// TIA Portal V17 export
// export: Created 2025-03-07T09:18:09.3594696Z, ExportSetting WithDefaults, DisplayName Totally Integrated Automation Portal, DisplayVersion V17 Update 8, DisplayName TIA Portal Openness, DisplayVersion V17 Update 8, DisplayName TIA Portal Version Control Interface, DisplayVersion V17, DisplayName SINAMICS Startdrive Advanced, DisplayVersion V17 SP2, DisplayName SINAMICS Startdrive G110M, G120, G120C, G120D, G120P, G115D, DisplayVersion V17 SP2, DisplayName SINAMICS Startdrive G130, G150, S120, S150, SINAMICS MV, S210, DisplayVersion V17 SP2, DisplayName STEP 7 Professional, DisplayVersion V17 Update 8, DisplayName SINUMERIK ONE STEP 7 Toolbox, DisplayVersion V17 Update 12, DisplayName SINUMERIK 840D sl STEP 7 Toolbox, DisplayVersion V17 Update 12, DisplayName STEP 7 Safety, DisplayVersion V17 Update 6, DisplayName WinCC Advanced, DisplayVersion V17 Update 8
FUNCTION "FC1251_PART_CYCLE_UNIT_02_CLADDING" : Void   // FC1251, LAD
{ S7_Optimized_Access := 'FALSE' }
AUTHOR : ETXETAR
VERSION : 1.0
// stored: AutoNumber false, IsIECCheckEnabled false, SetENOAutomatically false, UDAEnableTagReadback false
   VAR CONSTANT
      FC_NUMBER : DInt := 1251;
   END_VAR
   VAR_TEMP   // added for the SCL form of the ladder/FBD networks
      _w1 : Bool;
      _w2 : Bool;
      _w3 : Bool;
      _w4 : Bool;
   END_VAR
BEGIN

REGION Network 1: GENERAL CONDITIONS
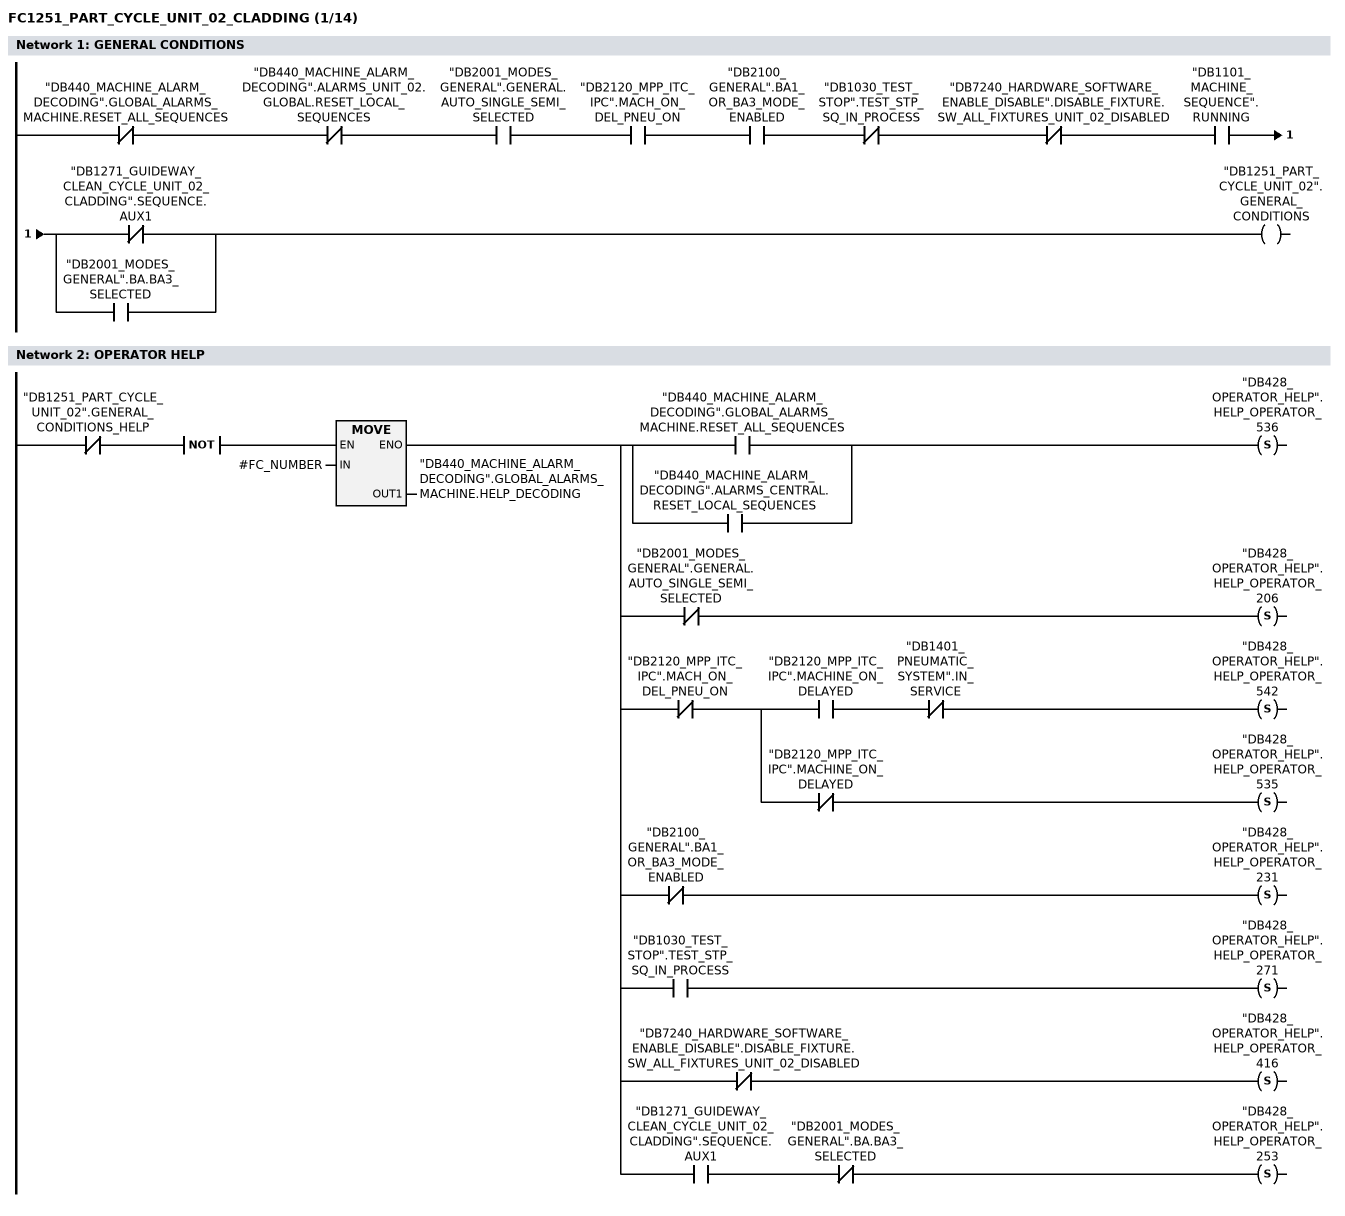
   RUNG wire#powerrail
      I_Contact( "DB440_MACHINE_ALARM_DECODING".GLOBAL_ALARMS_MACHINE.RESET_ALL_SEQUENCES )
      I_Contact( "DB440_MACHINE_ALARM_DECODING".ALARMS_UNIT_02.GLOBAL.RESET_LOCAL_SEQUENCES )
      Contact( "DB2001_MODES_GENERAL".GENERAL.AUTO_SINGLE_SEMI_SELECTED )
      Contact( "DB2120_MPP_ITC_IPC".MACH_ON_DEL_PNEU_ON )
      Contact( "DB2100_GENERAL".BA1_OR_BA3_MODE_ENABLED )
      I_Contact( "DB1030_TEST_STOP".TEST_STP_SQ_IN_PROCESS )
      I_Contact( "DB7240_HARDWARE_SOFTWARE_ENABLE_DISABLE".DISABLE_FIXTURE.SW_ALL_FIXTURES_UNIT_02_DISABLED )
      Contact( "DB1101_MACHINE_SEQUENCE".RUNNING )
      wire#w1
      I_Contact( "DB1271_GUIDEWAY_CLEAN_CYCLE_UNIT_02_CLADDING".SEQUENCE.AUX1 )
      wire#w2
      Coil( "DB1251_PART_CYCLE_UNIT_02".GENERAL_CONDITIONS )
   END_RUNG
   RUNG wire#w1
      Contact( "DB2001_MODES_GENERAL".BA.BA3_SELECTED )
   END_RUNG wire#w2
   // the same network as SCL:
   "DB1251_PART_CYCLE_UNIT_02".GENERAL_CONDITIONS := NOT "DB440_MACHINE_ALARM_DECODING".GLOBAL_ALARMS_MACHINE.RESET_ALL_SEQUENCES AND NOT "DB440_MACHINE_ALARM_DECODING".ALARMS_UNIT_02.GLOBAL.RESET_LOCAL_SEQUENCES AND "DB2001_MODES_GENERAL".GENERAL.AUTO_SINGLE_SEMI_SELECTED AND "DB2120_MPP_ITC_IPC".MACH_ON_DEL_PNEU_ON AND "DB2100_GENERAL".BA1_OR_BA3_MODE_ENABLED AND NOT "DB1030_TEST_STOP".TEST_STP_SQ_IN_PROCESS AND NOT "DB7240_HARDWARE_SOFTWARE_ENABLE_DISABLE".DISABLE_FIXTURE.SW_ALL_FIXTURES_UNIT_02_DISABLED AND "DB1101_MACHINE_SEQUENCE".RUNNING AND (NOT "DB1271_GUIDEWAY_CLEAN_CYCLE_UNIT_02_CLADDING".SEQUENCE.AUX1 OR "DB2001_MODES_GENERAL".BA.BA3_SELECTED);
END_REGION

REGION Network 2: OPERATOR HELP
   RUNG wire#powerrail
      I_Contact( "DB1251_PART_CYCLE_UNIT_02".GENERAL_CONDITIONS_HELP )
      Not()
      { S7_GenerateENO := "TRUE" } Move(in := #FC_NUMBER, out1 => "DB440_MACHINE_ALARM_DECODING".GLOBAL_ALARMS_MACHINE.HELP_DECODING)
      wire#w1
      Contact( "DB440_MACHINE_ALARM_DECODING".GLOBAL_ALARMS_MACHINE.RESET_ALL_SEQUENCES )
      wire#w2
      S_Coil( "DB428_OPERATOR_HELP".HELP_OPERATOR_536 )
   END_RUNG
   RUNG wire#w1
      Contact( "DB440_MACHINE_ALARM_DECODING".ALARMS_CENTRAL.RESET_LOCAL_SEQUENCES )
   END_RUNG wire#w2
   RUNG wire#w1
      I_Contact( "DB2001_MODES_GENERAL".GENERAL.AUTO_SINGLE_SEMI_SELECTED )
      S_Coil( "DB428_OPERATOR_HELP".HELP_OPERATOR_206 )
   END_RUNG
   RUNG wire#w1
      I_Contact( "DB2120_MPP_ITC_IPC".MACH_ON_DEL_PNEU_ON )
      wire#w3
      Contact( "DB2120_MPP_ITC_IPC".MACHINE_ON_DELAYED )
      I_Contact( "DB1401_PNEUMATIC_SYSTEM".IN_SERVICE )
      S_Coil( "DB428_OPERATOR_HELP".HELP_OPERATOR_542 )
   END_RUNG
   RUNG wire#w3
      I_Contact( "DB2120_MPP_ITC_IPC".MACHINE_ON_DELAYED )
      S_Coil( "DB428_OPERATOR_HELP".HELP_OPERATOR_535 )
   END_RUNG
   RUNG wire#w1
      I_Contact( "DB2100_GENERAL".BA1_OR_BA3_MODE_ENABLED )
      S_Coil( "DB428_OPERATOR_HELP".HELP_OPERATOR_231 )
   END_RUNG
   RUNG wire#w1
      Contact( "DB1030_TEST_STOP".TEST_STP_SQ_IN_PROCESS )
      S_Coil( "DB428_OPERATOR_HELP".HELP_OPERATOR_271 )
   END_RUNG
   RUNG wire#w1
      I_Contact( "DB7240_HARDWARE_SOFTWARE_ENABLE_DISABLE".DISABLE_FIXTURE.SW_ALL_FIXTURES_UNIT_02_DISABLED )
      S_Coil( "DB428_OPERATOR_HELP".HELP_OPERATOR_416 )
   END_RUNG
   RUNG wire#w1
      Contact( "DB1271_GUIDEWAY_CLEAN_CYCLE_UNIT_02_CLADDING".SEQUENCE.AUX1 )
      I_Contact( "DB2001_MODES_GENERAL".BA.BA3_SELECTED )
      S_Coil( "DB428_OPERATOR_HELP".HELP_OPERATOR_253 )
   END_RUNG
   // the same network as SCL:
   // ENO of a box is taken as its EN; it also drops when the box reports an error
   #_w1 := NOT (NOT "DB1251_PART_CYCLE_UNIT_02".GENERAL_CONDITIONS_HELP);
   IF #_w1 THEN "DB440_MACHINE_ALARM_DECODING".GLOBAL_ALARMS_MACHINE.HELP_DECODING := #FC_NUMBER; END_IF;
   IF #_w1 AND ("DB440_MACHINE_ALARM_DECODING".GLOBAL_ALARMS_MACHINE.RESET_ALL_SEQUENCES OR "DB440_MACHINE_ALARM_DECODING".ALARMS_CENTRAL.RESET_LOCAL_SEQUENCES) THEN
       "DB428_OPERATOR_HELP".HELP_OPERATOR_536 := TRUE;
   END_IF;
   IF #_w1 AND NOT "DB2001_MODES_GENERAL".GENERAL.AUTO_SINGLE_SEMI_SELECTED THEN
       "DB428_OPERATOR_HELP".HELP_OPERATOR_206 := TRUE;
   END_IF;
   #_w2 := #_w1 AND NOT "DB2120_MPP_ITC_IPC".MACH_ON_DEL_PNEU_ON;
   IF #_w2 AND "DB2120_MPP_ITC_IPC".MACHINE_ON_DELAYED AND NOT "DB1401_PNEUMATIC_SYSTEM".IN_SERVICE THEN
       "DB428_OPERATOR_HELP".HELP_OPERATOR_542 := TRUE;
   END_IF;
   IF #_w2 AND NOT "DB2120_MPP_ITC_IPC".MACHINE_ON_DELAYED THEN
       "DB428_OPERATOR_HELP".HELP_OPERATOR_535 := TRUE;
   END_IF;
   IF #_w1 AND NOT "DB2100_GENERAL".BA1_OR_BA3_MODE_ENABLED THEN
       "DB428_OPERATOR_HELP".HELP_OPERATOR_231 := TRUE;
   END_IF;
   IF #_w1 AND "DB1030_TEST_STOP".TEST_STP_SQ_IN_PROCESS THEN
       "DB428_OPERATOR_HELP".HELP_OPERATOR_271 := TRUE;
   END_IF;
   IF #_w1 AND NOT "DB7240_HARDWARE_SOFTWARE_ENABLE_DISABLE".DISABLE_FIXTURE.SW_ALL_FIXTURES_UNIT_02_DISABLED THEN
       "DB428_OPERATOR_HELP".HELP_OPERATOR_416 := TRUE;
   END_IF;
   IF #_w1 AND "DB1271_GUIDEWAY_CLEAN_CYCLE_UNIT_02_CLADDING".SEQUENCE.AUX1 AND NOT "DB2001_MODES_GENERAL".BA.BA3_SELECTED THEN
       "DB428_OPERATOR_HELP".HELP_OPERATOR_253 := TRUE;
   END_IF;
END_REGION

REGION Network 3: INITIAL CONDITIONS
   // CAMBIAR LOS BITS DE QUALITY CUANDO ESTEN HECHOS
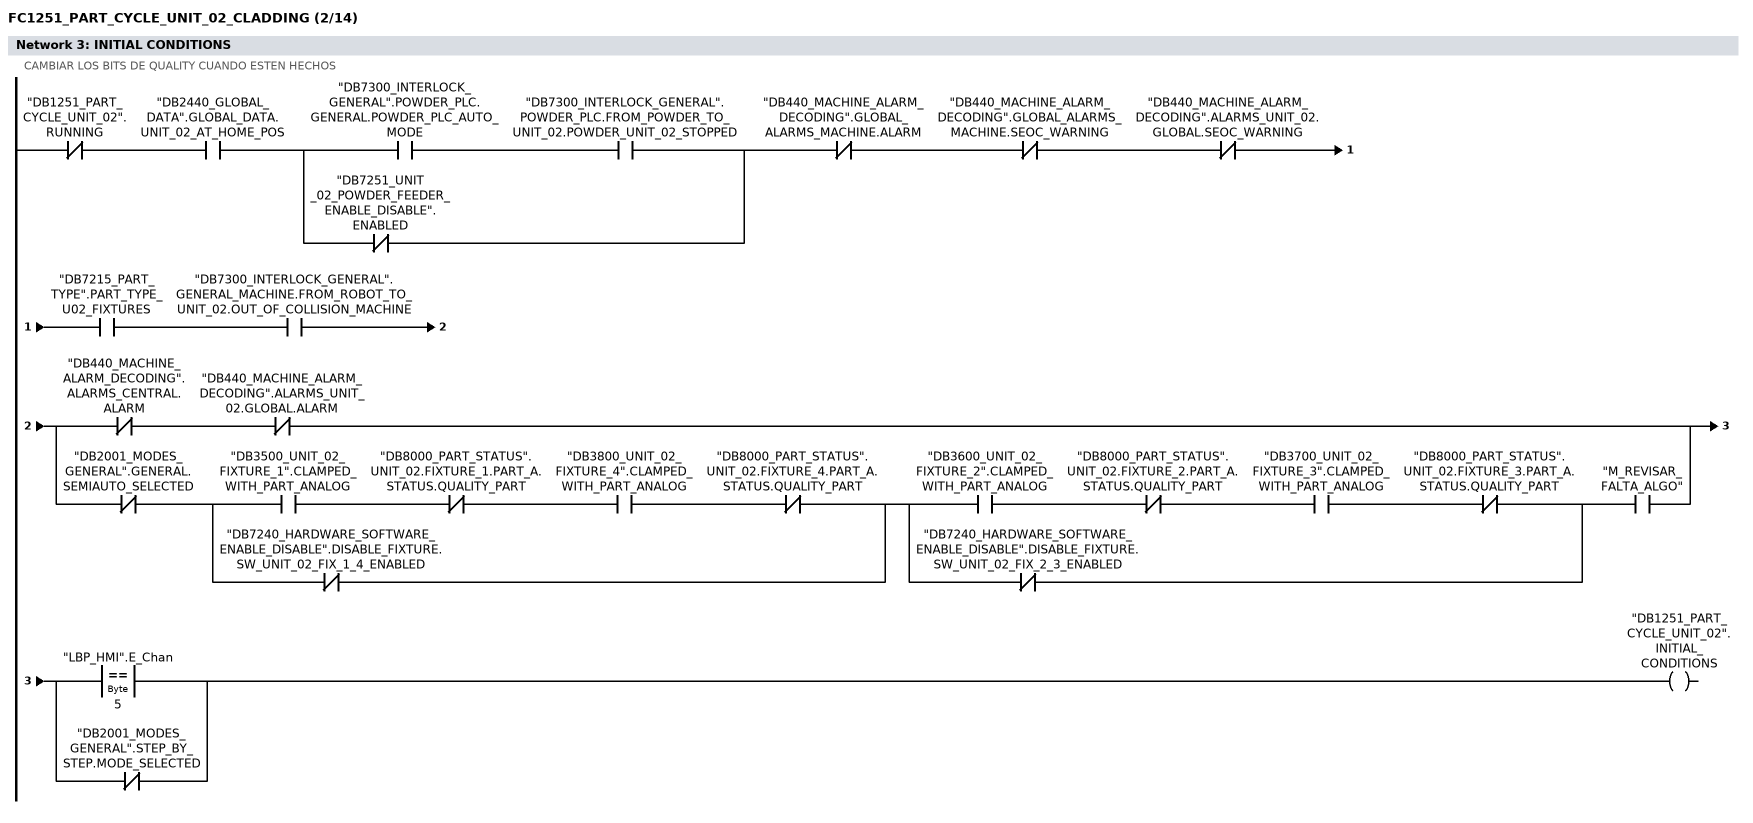
   RUNG wire#powerrail
      I_Contact( "DB1251_PART_CYCLE_UNIT_02".RUNNING )
      Contact( "DB2440_GLOBAL_DATA".GLOBAL_DATA.UNIT_02_AT_HOME_POS )
      wire#w1
      Contact( "DB7300_INTERLOCK_GENERAL".POWDER_PLC.GENERAL.POWDER_PLC_AUTO_MODE )
      Contact( "DB7300_INTERLOCK_GENERAL".POWDER_PLC.FROM_POWDER_TO_UNIT_02.POWDER_UNIT_02_STOPPED )
      wire#w2
      I_Contact( "DB440_MACHINE_ALARM_DECODING".GLOBAL_ALARMS_MACHINE.ALARM )
      I_Contact( "DB440_MACHINE_ALARM_DECODING".GLOBAL_ALARMS_MACHINE.SEOC_WARNING )
      I_Contact( "DB440_MACHINE_ALARM_DECODING".ALARMS_UNIT_02.GLOBAL.SEOC_WARNING )
      Contact( "DB7215_PART_TYPE".PART_TYPE_U02_FIXTURES )
      Contact( "DB7300_INTERLOCK_GENERAL".GENERAL_MACHINE.FROM_ROBOT_TO_UNIT_02.OUT_OF_COLLISION_MACHINE )
      wire#w3
      I_Contact( "DB440_MACHINE_ALARM_DECODING".ALARMS_CENTRAL.ALARM )
      I_Contact( "DB440_MACHINE_ALARM_DECODING".ALARMS_UNIT_02.GLOBAL.ALARM )
      wire#w4
      { S7_Templates := "SrcType := Byte" } EQ_Contact(in1 := "LBP_HMI".E_Chan, in2 := 5)
      wire#w8
      Coil( "DB1251_PART_CYCLE_UNIT_02".INITIAL_CONDITIONS )
   END_RUNG
   RUNG wire#w1
      I_Contact( "DB7251_UNIT _02_POWDER_FEEDER_ENABLE_DISABLE".ENABLED )
   END_RUNG wire#w2
   RUNG wire#w3
      I_Contact( "DB2001_MODES_GENERAL".GENERAL.SEMIAUTO_SELECTED )
      wire#w5
      Contact( "DB3500_UNIT_02_FIXTURE_1".CLAMPED_WITH_PART_ANALOG )
      I_Contact( "DB8000_PART_STATUS".UNIT_02.FIXTURE_1.PART_A.STATUS.QUALITY_PART )
      Contact( "DB3800_UNIT_02_FIXTURE_4".CLAMPED_WITH_PART_ANALOG )
      I_Contact( "DB8000_PART_STATUS".UNIT_02.FIXTURE_4.PART_A.STATUS.QUALITY_PART )
      wire#w6
      Contact( "DB3600_UNIT_02_FIXTURE_2".CLAMPED_WITH_PART_ANALOG )
      I_Contact( "DB8000_PART_STATUS".UNIT_02.FIXTURE_2.PART_A.STATUS.QUALITY_PART )
      Contact( "DB3700_UNIT_02_FIXTURE_3".CLAMPED_WITH_PART_ANALOG )
      I_Contact( "DB8000_PART_STATUS".UNIT_02.FIXTURE_3.PART_A.STATUS.QUALITY_PART )
      wire#w7
      Contact( "M_REVISAR_FALTA_ALGO" )
   END_RUNG wire#w4
   RUNG wire#w5
      I_Contact( "DB7240_HARDWARE_SOFTWARE_ENABLE_DISABLE".DISABLE_FIXTURE.SW_UNIT_02_FIX_1_4_ENABLED )
   END_RUNG wire#w6
   RUNG wire#w6
      I_Contact( "DB7240_HARDWARE_SOFTWARE_ENABLE_DISABLE".DISABLE_FIXTURE.SW_UNIT_02_FIX_2_3_ENABLED )
   END_RUNG wire#w7
   RUNG wire#w4
      I_Contact( "DB2001_MODES_GENERAL".STEP_BY_STEP.MODE_SELECTED )
   END_RUNG wire#w8
   // the same network as SCL:
   "DB1251_PART_CYCLE_UNIT_02".INITIAL_CONDITIONS := NOT "DB1251_PART_CYCLE_UNIT_02".RUNNING AND "DB2440_GLOBAL_DATA".GLOBAL_DATA.UNIT_02_AT_HOME_POS AND (("DB7300_INTERLOCK_GENERAL".POWDER_PLC.GENERAL.POWDER_PLC_AUTO_MODE AND "DB7300_INTERLOCK_GENERAL".POWDER_PLC.FROM_POWDER_TO_UNIT_02.POWDER_UNIT_02_STOPPED) OR NOT "DB7251_UNIT _02_POWDER_FEEDER_ENABLE_DISABLE".ENABLED) AND NOT "DB440_MACHINE_ALARM_DECODING".GLOBAL_ALARMS_MACHINE.ALARM AND NOT "DB440_MACHINE_ALARM_DECODING".GLOBAL_ALARMS_MACHINE.SEOC_WARNING AND NOT "DB440_MACHINE_ALARM_DECODING".ALARMS_UNIT_02.GLOBAL.SEOC_WARNING AND "DB7215_PART_TYPE".PART_TYPE_U02_FIXTURES AND "DB7300_INTERLOCK_GENERAL".GENERAL_MACHINE.FROM_ROBOT_TO_UNIT_02.OUT_OF_COLLISION_MACHINE AND ((NOT "DB440_MACHINE_ALARM_DECODING".ALARMS_CENTRAL.ALARM AND NOT "DB440_MACHINE_ALARM_DECODING".ALARMS_UNIT_02.GLOBAL.ALARM) OR (NOT "DB2001_MODES_GENERAL".GENERAL.SEMIAUTO_SELECTED AND (("DB3500_UNIT_02_FIXTURE_1".CLAMPED_WITH_PART_ANALOG AND NOT "DB8000_PART_STATUS".UNIT_02.FIXTURE_1.PART_A.STATUS.QUALITY_PART AND "DB3800_UNIT_02_FIXTURE_4".CLAMPED_WITH_PART_ANALOG AND NOT "DB8000_PART_STATUS".UNIT_02.FIXTURE_4.PART_A.STATUS.QUALITY_PART) OR NOT "DB7240_HARDWARE_SOFTWARE_ENABLE_DISABLE".DISABLE_FIXTURE.SW_UNIT_02_FIX_1_4_ENABLED) AND (("DB3600_UNIT_02_FIXTURE_2".CLAMPED_WITH_PART_ANALOG AND NOT "DB8000_PART_STATUS".UNIT_02.FIXTURE_2.PART_A.STATUS.QUALITY_PART AND "DB3700_UNIT_02_FIXTURE_3".CLAMPED_WITH_PART_ANALOG AND NOT "DB8000_PART_STATUS".UNIT_02.FIXTURE_3.PART_A.STATUS.QUALITY_PART) OR NOT "DB7240_HARDWARE_SOFTWARE_ENABLE_DISABLE".DISABLE_FIXTURE.SW_UNIT_02_FIX_2_3_ENABLED) AND "M_REVISAR_FALTA_ALGO")) AND (("LBP_HMI".E_Chan = 5) OR NOT "DB2001_MODES_GENERAL".STEP_BY_STEP.MODE_SELECTED);
END_REGION

REGION Network 4: OPERATOR HELP
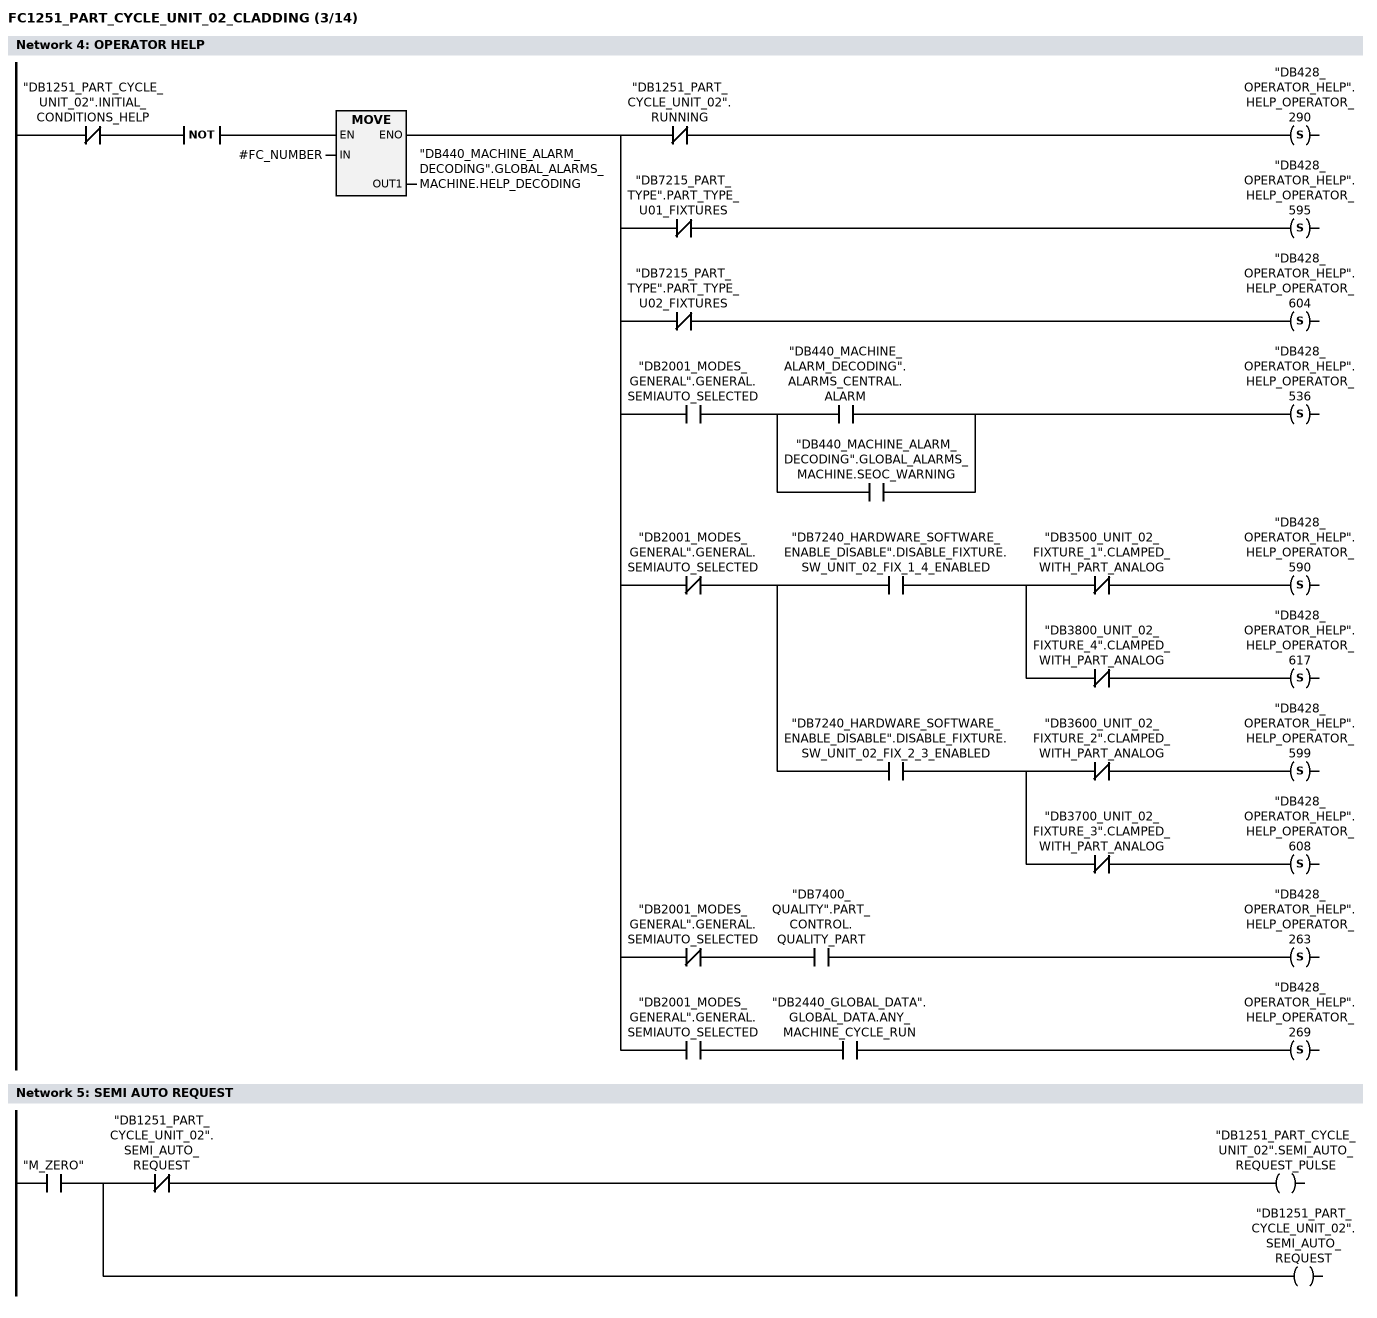
   RUNG wire#powerrail
      I_Contact( "DB1251_PART_CYCLE_UNIT_02".INITIAL_CONDITIONS_HELP )
      Not()
      { S7_GenerateENO := "TRUE" } Move(in := #FC_NUMBER, out1 => "DB440_MACHINE_ALARM_DECODING".GLOBAL_ALARMS_MACHINE.HELP_DECODING)
      wire#w1
      I_Contact( "DB1251_PART_CYCLE_UNIT_02".RUNNING )
      S_Coil( "DB428_OPERATOR_HELP".HELP_OPERATOR_290 )
   END_RUNG
   RUNG wire#w1
      I_Contact( "DB7215_PART_TYPE".PART_TYPE_U01_FIXTURES )
      S_Coil( "DB428_OPERATOR_HELP".HELP_OPERATOR_595 )
   END_RUNG
   RUNG wire#w1
      I_Contact( "DB7215_PART_TYPE".PART_TYPE_U02_FIXTURES )
      S_Coil( "DB428_OPERATOR_HELP".HELP_OPERATOR_604 )
   END_RUNG
   RUNG wire#w1
      Contact( "DB2001_MODES_GENERAL".GENERAL.SEMIAUTO_SELECTED )
      wire#w2
      Contact( "DB440_MACHINE_ALARM_DECODING".ALARMS_CENTRAL.ALARM )
      wire#w3
      S_Coil( "DB428_OPERATOR_HELP".HELP_OPERATOR_536 )
   END_RUNG
   RUNG wire#w2
      Contact( "DB440_MACHINE_ALARM_DECODING".GLOBAL_ALARMS_MACHINE.SEOC_WARNING )
   END_RUNG wire#w3
   RUNG wire#w1
      I_Contact( "DB2001_MODES_GENERAL".GENERAL.SEMIAUTO_SELECTED )
      wire#w4
      Contact( "DB7240_HARDWARE_SOFTWARE_ENABLE_DISABLE".DISABLE_FIXTURE.SW_UNIT_02_FIX_1_4_ENABLED )
      wire#w5
      I_Contact( "DB3500_UNIT_02_FIXTURE_1".CLAMPED_WITH_PART_ANALOG )
      S_Coil( "DB428_OPERATOR_HELP".HELP_OPERATOR_590 )
   END_RUNG
   RUNG wire#w5
      I_Contact( "DB3800_UNIT_02_FIXTURE_4".CLAMPED_WITH_PART_ANALOG )
      S_Coil( "DB428_OPERATOR_HELP".HELP_OPERATOR_617 )
   END_RUNG
   RUNG wire#w4
      Contact( "DB7240_HARDWARE_SOFTWARE_ENABLE_DISABLE".DISABLE_FIXTURE.SW_UNIT_02_FIX_2_3_ENABLED )
      wire#w6
      I_Contact( "DB3600_UNIT_02_FIXTURE_2".CLAMPED_WITH_PART_ANALOG )
      S_Coil( "DB428_OPERATOR_HELP".HELP_OPERATOR_599 )
   END_RUNG
   RUNG wire#w6
      I_Contact( "DB3700_UNIT_02_FIXTURE_3".CLAMPED_WITH_PART_ANALOG )
      S_Coil( "DB428_OPERATOR_HELP".HELP_OPERATOR_608 )
   END_RUNG
   RUNG wire#w1
      I_Contact( "DB2001_MODES_GENERAL".GENERAL.SEMIAUTO_SELECTED )
      Contact( "DB7400_QUALITY".PART_CONTROL.QUALITY_PART )
      S_Coil( "DB428_OPERATOR_HELP".HELP_OPERATOR_263 )
   END_RUNG
   RUNG wire#w1
      Contact( "DB2001_MODES_GENERAL".GENERAL.SEMIAUTO_SELECTED )
      Contact( "DB2440_GLOBAL_DATA".GLOBAL_DATA.ANY_MACHINE_CYCLE_RUN )
      S_Coil( "DB428_OPERATOR_HELP".HELP_OPERATOR_269 )
   END_RUNG
   // the same network as SCL:
   // ENO of a box is taken as its EN; it also drops when the box reports an error
   #_w1 := NOT (NOT "DB1251_PART_CYCLE_UNIT_02".INITIAL_CONDITIONS_HELP);
   IF #_w1 THEN "DB440_MACHINE_ALARM_DECODING".GLOBAL_ALARMS_MACHINE.HELP_DECODING := #FC_NUMBER; END_IF;
   IF #_w1 AND NOT "DB1251_PART_CYCLE_UNIT_02".RUNNING THEN
       "DB428_OPERATOR_HELP".HELP_OPERATOR_290 := TRUE;
   END_IF;
   IF #_w1 AND NOT "DB7215_PART_TYPE".PART_TYPE_U01_FIXTURES THEN
       "DB428_OPERATOR_HELP".HELP_OPERATOR_595 := TRUE;
   END_IF;
   IF #_w1 AND NOT "DB7215_PART_TYPE".PART_TYPE_U02_FIXTURES THEN
       "DB428_OPERATOR_HELP".HELP_OPERATOR_604 := TRUE;
   END_IF;
   IF #_w1 AND "DB2001_MODES_GENERAL".GENERAL.SEMIAUTO_SELECTED AND ("DB440_MACHINE_ALARM_DECODING".ALARMS_CENTRAL.ALARM OR "DB440_MACHINE_ALARM_DECODING".GLOBAL_ALARMS_MACHINE.SEOC_WARNING) THEN
       "DB428_OPERATOR_HELP".HELP_OPERATOR_536 := TRUE;
   END_IF;
   #_w2 := #_w1 AND NOT "DB2001_MODES_GENERAL".GENERAL.SEMIAUTO_SELECTED;
   #_w3 := #_w2 AND "DB7240_HARDWARE_SOFTWARE_ENABLE_DISABLE".DISABLE_FIXTURE.SW_UNIT_02_FIX_1_4_ENABLED;
   IF #_w3 AND NOT "DB3500_UNIT_02_FIXTURE_1".CLAMPED_WITH_PART_ANALOG THEN
       "DB428_OPERATOR_HELP".HELP_OPERATOR_590 := TRUE;
   END_IF;
   IF #_w3 AND NOT "DB3800_UNIT_02_FIXTURE_4".CLAMPED_WITH_PART_ANALOG THEN
       "DB428_OPERATOR_HELP".HELP_OPERATOR_617 := TRUE;
   END_IF;
   #_w4 := #_w2 AND "DB7240_HARDWARE_SOFTWARE_ENABLE_DISABLE".DISABLE_FIXTURE.SW_UNIT_02_FIX_2_3_ENABLED;
   IF #_w4 AND NOT "DB3600_UNIT_02_FIXTURE_2".CLAMPED_WITH_PART_ANALOG THEN
       "DB428_OPERATOR_HELP".HELP_OPERATOR_599 := TRUE;
   END_IF;
   IF #_w4 AND NOT "DB3700_UNIT_02_FIXTURE_3".CLAMPED_WITH_PART_ANALOG THEN
       "DB428_OPERATOR_HELP".HELP_OPERATOR_608 := TRUE;
   END_IF;
   IF #_w1 AND NOT "DB2001_MODES_GENERAL".GENERAL.SEMIAUTO_SELECTED AND "DB7400_QUALITY".PART_CONTROL.QUALITY_PART THEN
       "DB428_OPERATOR_HELP".HELP_OPERATOR_263 := TRUE;
   END_IF;
   IF #_w1 AND "DB2001_MODES_GENERAL".GENERAL.SEMIAUTO_SELECTED AND "DB2440_GLOBAL_DATA".GLOBAL_DATA.ANY_MACHINE_CYCLE_RUN THEN
       "DB428_OPERATOR_HELP".HELP_OPERATOR_269 := TRUE;
   END_IF;
END_REGION

REGION Network 5: SEMI AUTO REQUEST
   RUNG wire#powerrail
      Contact( "M_ZERO" )
      wire#w1
      I_Contact( "DB1251_PART_CYCLE_UNIT_02".SEMI_AUTO_REQUEST )
      Coil( "DB1251_PART_CYCLE_UNIT_02".SEMI_AUTO_REQUEST_PULSE )
   END_RUNG
   RUNG wire#w1
      Coil( "DB1251_PART_CYCLE_UNIT_02".SEMI_AUTO_REQUEST )
   END_RUNG
   // the same network as SCL:
   "DB1251_PART_CYCLE_UNIT_02".SEMI_AUTO_REQUEST_PULSE := "M_ZERO" AND NOT "DB1251_PART_CYCLE_UNIT_02".SEMI_AUTO_REQUEST;
   "DB1251_PART_CYCLE_UNIT_02".SEMI_AUTO_REQUEST := "M_ZERO";
END_REGION

REGION Network 6: OPERATOR HELP
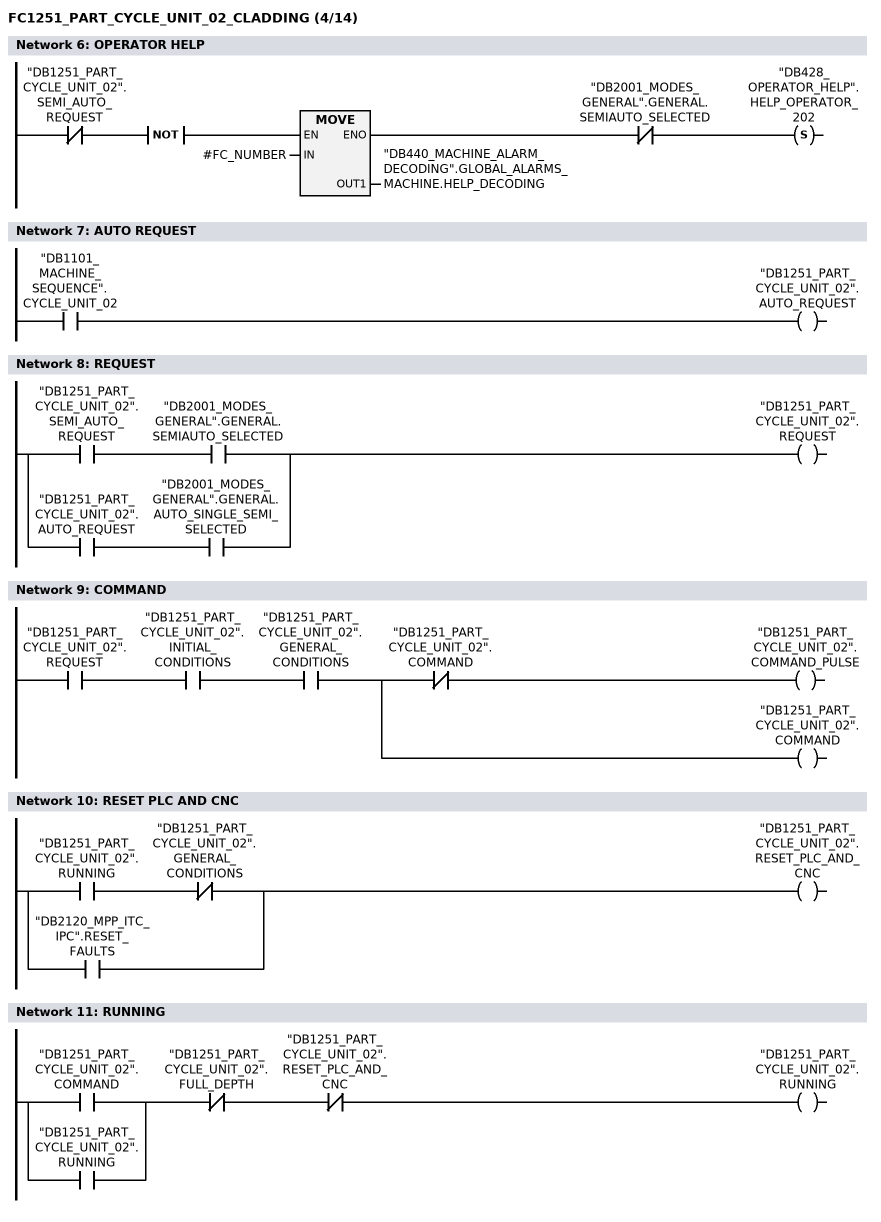
   RUNG wire#powerrail
      I_Contact( "DB1251_PART_CYCLE_UNIT_02".SEMI_AUTO_REQUEST )
      Not()
      { S7_GenerateENO := "TRUE" } Move(in := #FC_NUMBER, out1 => "DB440_MACHINE_ALARM_DECODING".GLOBAL_ALARMS_MACHINE.HELP_DECODING)
      I_Contact( "DB2001_MODES_GENERAL".GENERAL.SEMIAUTO_SELECTED )
      S_Coil( "DB428_OPERATOR_HELP".HELP_OPERATOR_202 )
   END_RUNG
   // the same network as SCL:
   // ENO of a box is taken as its EN; it also drops when the box reports an error
   #_w1 := NOT (NOT "DB1251_PART_CYCLE_UNIT_02".SEMI_AUTO_REQUEST);
   IF #_w1 THEN "DB440_MACHINE_ALARM_DECODING".GLOBAL_ALARMS_MACHINE.HELP_DECODING := #FC_NUMBER; END_IF;
   IF #_w1 AND NOT "DB2001_MODES_GENERAL".GENERAL.SEMIAUTO_SELECTED THEN
       "DB428_OPERATOR_HELP".HELP_OPERATOR_202 := TRUE;
   END_IF;
END_REGION

REGION Network 7: AUTO REQUEST
   RUNG wire#powerrail
      Contact( "DB1101_MACHINE_SEQUENCE".CYCLE_UNIT_02 )
      Coil( "DB1251_PART_CYCLE_UNIT_02".AUTO_REQUEST )
   END_RUNG
   // the same network as SCL:
   "DB1251_PART_CYCLE_UNIT_02".AUTO_REQUEST := "DB1101_MACHINE_SEQUENCE".CYCLE_UNIT_02;
END_REGION

REGION Network 8: REQUEST
   RUNG wire#powerrail
      Contact( "DB1251_PART_CYCLE_UNIT_02".SEMI_AUTO_REQUEST )
      Contact( "DB2001_MODES_GENERAL".GENERAL.SEMIAUTO_SELECTED )
      wire#w1
      Coil( "DB1251_PART_CYCLE_UNIT_02".REQUEST )
   END_RUNG
   RUNG wire#powerrail
      Contact( "DB1251_PART_CYCLE_UNIT_02".AUTO_REQUEST )
      Contact( "DB2001_MODES_GENERAL".GENERAL.AUTO_SINGLE_SEMI_SELECTED )
   END_RUNG wire#w1
   // the same network as SCL:
   "DB1251_PART_CYCLE_UNIT_02".REQUEST := ("DB1251_PART_CYCLE_UNIT_02".SEMI_AUTO_REQUEST AND "DB2001_MODES_GENERAL".GENERAL.SEMIAUTO_SELECTED) OR ("DB1251_PART_CYCLE_UNIT_02".AUTO_REQUEST AND "DB2001_MODES_GENERAL".GENERAL.AUTO_SINGLE_SEMI_SELECTED);
END_REGION

REGION Network 9: COMMAND
   RUNG wire#powerrail
      Contact( "DB1251_PART_CYCLE_UNIT_02".REQUEST )
      Contact( "DB1251_PART_CYCLE_UNIT_02".INITIAL_CONDITIONS )
      Contact( "DB1251_PART_CYCLE_UNIT_02".GENERAL_CONDITIONS )
      wire#w1
      I_Contact( "DB1251_PART_CYCLE_UNIT_02".COMMAND )
      Coil( "DB1251_PART_CYCLE_UNIT_02".COMMAND_PULSE )
   END_RUNG
   RUNG wire#w1
      Coil( "DB1251_PART_CYCLE_UNIT_02".COMMAND )
   END_RUNG
   // the same network as SCL:
   #_w1 := "DB1251_PART_CYCLE_UNIT_02".REQUEST AND "DB1251_PART_CYCLE_UNIT_02".INITIAL_CONDITIONS AND "DB1251_PART_CYCLE_UNIT_02".GENERAL_CONDITIONS;
   "DB1251_PART_CYCLE_UNIT_02".COMMAND_PULSE := #_w1 AND NOT "DB1251_PART_CYCLE_UNIT_02".COMMAND;
   "DB1251_PART_CYCLE_UNIT_02".COMMAND := #_w1;
END_REGION

REGION Network 10: RESET PLC AND CNC
   RUNG wire#powerrail
      Contact( "DB1251_PART_CYCLE_UNIT_02".RUNNING )
      I_Contact( "DB1251_PART_CYCLE_UNIT_02".GENERAL_CONDITIONS )
      wire#w1
      Coil( "DB1251_PART_CYCLE_UNIT_02".RESET_PLC_AND_CNC )
   END_RUNG
   RUNG wire#powerrail
      Contact( "DB2120_MPP_ITC_IPC".RESET_FAULTS )
   END_RUNG wire#w1
   // the same network as SCL:
   "DB1251_PART_CYCLE_UNIT_02".RESET_PLC_AND_CNC := ("DB1251_PART_CYCLE_UNIT_02".RUNNING AND NOT "DB1251_PART_CYCLE_UNIT_02".GENERAL_CONDITIONS) OR "DB2120_MPP_ITC_IPC".RESET_FAULTS;
END_REGION

REGION Network 11: RUNNING
   RUNG wire#powerrail
      Contact( "DB1251_PART_CYCLE_UNIT_02".COMMAND )
      wire#w1
      I_Contact( "DB1251_PART_CYCLE_UNIT_02".FULL_DEPTH )
      I_Contact( "DB1251_PART_CYCLE_UNIT_02".RESET_PLC_AND_CNC )
      Coil( "DB1251_PART_CYCLE_UNIT_02".RUNNING )
   END_RUNG
   RUNG wire#powerrail
      Contact( "DB1251_PART_CYCLE_UNIT_02".RUNNING )
   END_RUNG wire#w1
   // the same network as SCL:
   "DB1251_PART_CYCLE_UNIT_02".RUNNING := ("DB1251_PART_CYCLE_UNIT_02".COMMAND OR "DB1251_PART_CYCLE_UNIT_02".RUNNING) AND NOT "DB1251_PART_CYCLE_UNIT_02".FULL_DEPTH AND NOT "DB1251_PART_CYCLE_UNIT_02".RESET_PLC_AND_CNC;
END_REGION

REGION Network 12: UNIT 02 STATION 1 CONDITIONS OK FOR STATION 0 CYCLE REQUEST
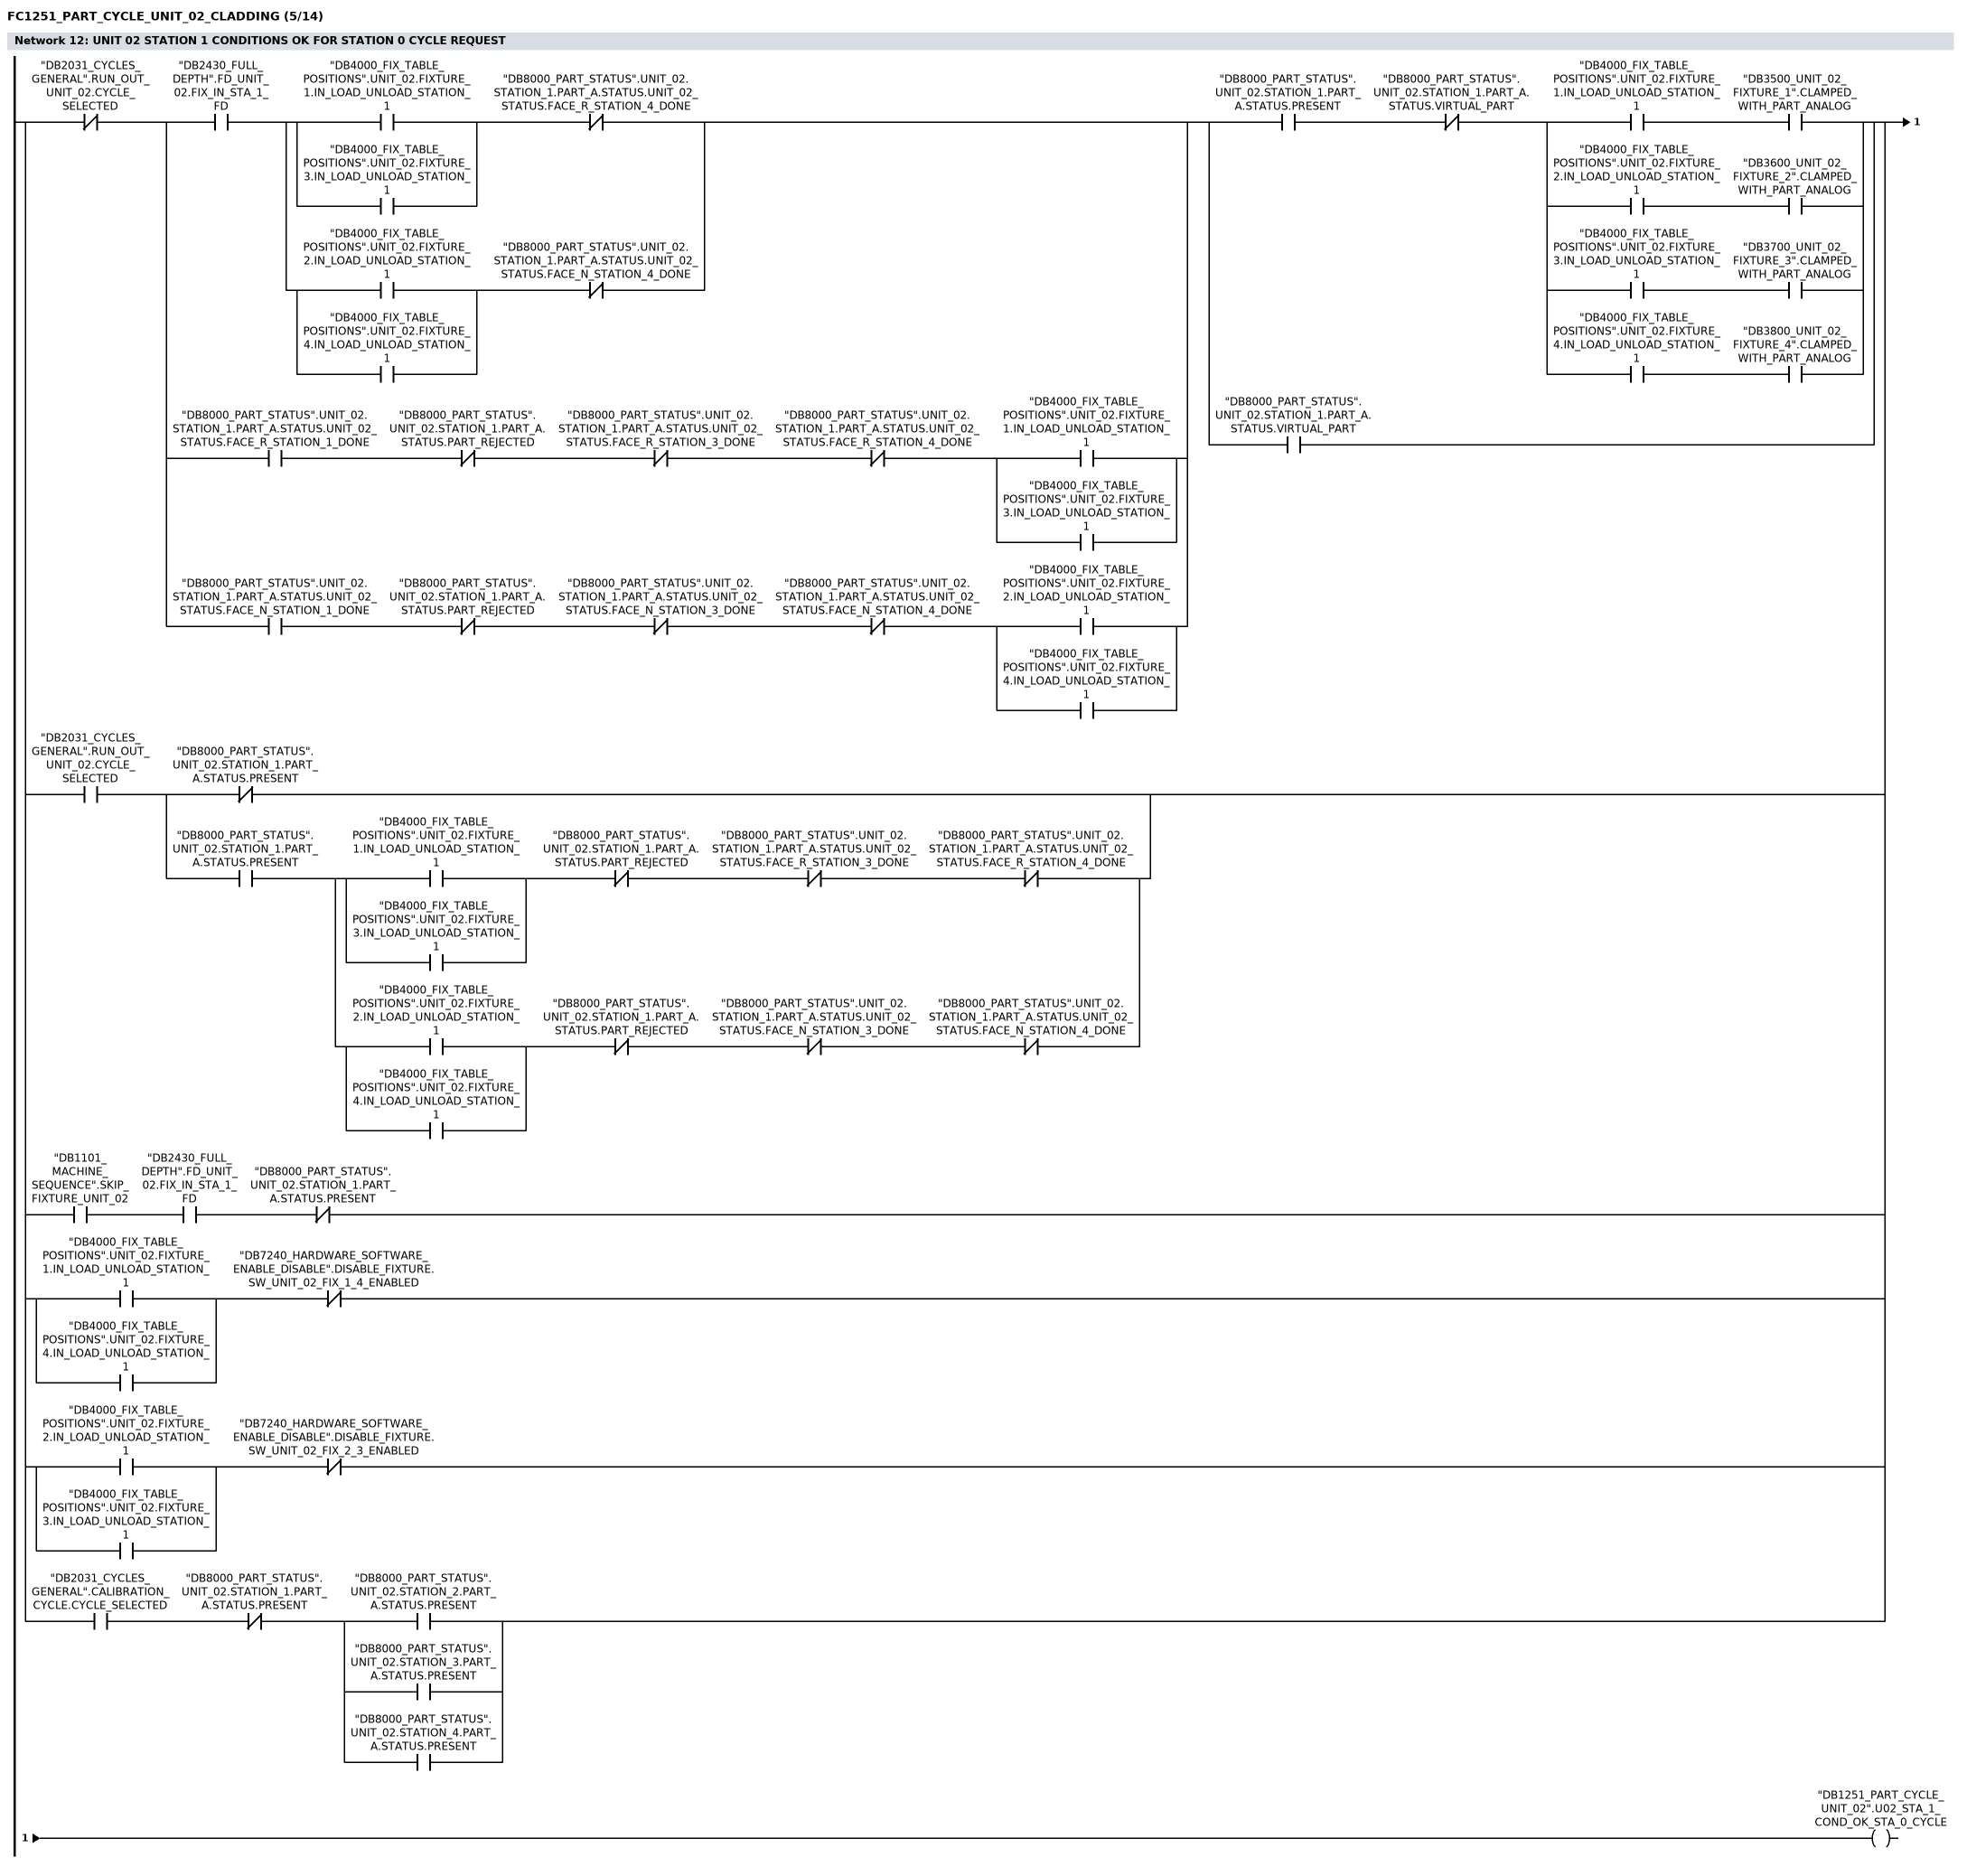
   RUNG wire#powerrail
      I_Contact( "DB2031_CYCLES_GENERAL".RUN_OUT_UNIT_02.CYCLE_SELECTED )
      wire#w1
      Contact( "DB2430_FULL_DEPTH".FD_UNIT_02.FIX_IN_STA_1_FD )
      wire#w2
      Contact( "DB4000_FIX_TABLE_POSITIONS".UNIT_02.FIXTURE_1.IN_LOAD_UNLOAD_STATION_1 )
      wire#w3
      I_Contact( "DB8000_PART_STATUS".UNIT_02.STATION_1.PART_A.STATUS.UNIT_02_STATUS.FACE_R_STATION_4_DONE )
      wire#w4
      Contact( "DB8000_PART_STATUS".UNIT_02.STATION_1.PART_A.STATUS.PRESENT )
      I_Contact( "DB8000_PART_STATUS".UNIT_02.STATION_1.PART_A.STATUS.VIRTUAL_PART )
      wire#w8
      Contact( "DB4000_FIX_TABLE_POSITIONS".UNIT_02.FIXTURE_1.IN_LOAD_UNLOAD_STATION_1 )
      Contact( "DB3500_UNIT_02_FIXTURE_1".CLAMPED_WITH_PART_ANALOG )
      wire#w9
      Coil( "DB1251_PART_CYCLE_UNIT_02".U02_STA_1_COND_OK_STA_0_CYCLE )
   END_RUNG
   RUNG wire#w2
      Contact( "DB4000_FIX_TABLE_POSITIONS".UNIT_02.FIXTURE_3.IN_LOAD_UNLOAD_STATION_1 )
   END_RUNG wire#w3
   RUNG wire#w2
      Contact( "DB4000_FIX_TABLE_POSITIONS".UNIT_02.FIXTURE_2.IN_LOAD_UNLOAD_STATION_1 )
      wire#w5
      I_Contact( "DB8000_PART_STATUS".UNIT_02.STATION_1.PART_A.STATUS.UNIT_02_STATUS.FACE_N_STATION_4_DONE )
   END_RUNG wire#w4
   RUNG wire#w2
      Contact( "DB4000_FIX_TABLE_POSITIONS".UNIT_02.FIXTURE_4.IN_LOAD_UNLOAD_STATION_1 )
   END_RUNG wire#w5
   RUNG wire#w1
      Contact( "DB8000_PART_STATUS".UNIT_02.STATION_1.PART_A.STATUS.UNIT_02_STATUS.FACE_R_STATION_1_DONE )
      I_Contact( "DB8000_PART_STATUS".UNIT_02.STATION_1.PART_A.STATUS.PART_REJECTED )
      I_Contact( "DB8000_PART_STATUS".UNIT_02.STATION_1.PART_A.STATUS.UNIT_02_STATUS.FACE_R_STATION_3_DONE )
      I_Contact( "DB8000_PART_STATUS".UNIT_02.STATION_1.PART_A.STATUS.UNIT_02_STATUS.FACE_R_STATION_4_DONE )
      wire#w6
      Contact( "DB4000_FIX_TABLE_POSITIONS".UNIT_02.FIXTURE_1.IN_LOAD_UNLOAD_STATION_1 )
   END_RUNG wire#w4
   RUNG wire#w6
      Contact( "DB4000_FIX_TABLE_POSITIONS".UNIT_02.FIXTURE_3.IN_LOAD_UNLOAD_STATION_1 )
   END_RUNG wire#w4
   RUNG wire#w1
      Contact( "DB8000_PART_STATUS".UNIT_02.STATION_1.PART_A.STATUS.UNIT_02_STATUS.FACE_N_STATION_1_DONE )
      I_Contact( "DB8000_PART_STATUS".UNIT_02.STATION_1.PART_A.STATUS.PART_REJECTED )
      I_Contact( "DB8000_PART_STATUS".UNIT_02.STATION_1.PART_A.STATUS.UNIT_02_STATUS.FACE_N_STATION_3_DONE )
      I_Contact( "DB8000_PART_STATUS".UNIT_02.STATION_1.PART_A.STATUS.UNIT_02_STATUS.FACE_N_STATION_4_DONE )
      wire#w7
      Contact( "DB4000_FIX_TABLE_POSITIONS".UNIT_02.FIXTURE_2.IN_LOAD_UNLOAD_STATION_1 )
   END_RUNG wire#w4
   RUNG wire#w7
      Contact( "DB4000_FIX_TABLE_POSITIONS".UNIT_02.FIXTURE_4.IN_LOAD_UNLOAD_STATION_1 )
   END_RUNG wire#w4
   RUNG wire#w8
      Contact( "DB4000_FIX_TABLE_POSITIONS".UNIT_02.FIXTURE_2.IN_LOAD_UNLOAD_STATION_1 )
      Contact( "DB3600_UNIT_02_FIXTURE_2".CLAMPED_WITH_PART_ANALOG )
   END_RUNG wire#w9
   RUNG wire#w8
      Contact( "DB4000_FIX_TABLE_POSITIONS".UNIT_02.FIXTURE_3.IN_LOAD_UNLOAD_STATION_1 )
      Contact( "DB3700_UNIT_02_FIXTURE_3".CLAMPED_WITH_PART_ANALOG )
   END_RUNG wire#w9
   RUNG wire#w8
      Contact( "DB4000_FIX_TABLE_POSITIONS".UNIT_02.FIXTURE_4.IN_LOAD_UNLOAD_STATION_1 )
      Contact( "DB3800_UNIT_02_FIXTURE_4".CLAMPED_WITH_PART_ANALOG )
   END_RUNG wire#w9
   RUNG wire#w4
      Contact( "DB8000_PART_STATUS".UNIT_02.STATION_1.PART_A.STATUS.VIRTUAL_PART )
   END_RUNG wire#w9
   RUNG wire#powerrail
      Contact( "DB2031_CYCLES_GENERAL".RUN_OUT_UNIT_02.CYCLE_SELECTED )
      wire#w10
      I_Contact( "DB8000_PART_STATUS".UNIT_02.STATION_1.PART_A.STATUS.PRESENT )
   END_RUNG wire#w9
   RUNG wire#w10
      Contact( "DB8000_PART_STATUS".UNIT_02.STATION_1.PART_A.STATUS.PRESENT )
      wire#w11
      Contact( "DB4000_FIX_TABLE_POSITIONS".UNIT_02.FIXTURE_1.IN_LOAD_UNLOAD_STATION_1 )
      wire#w12
      I_Contact( "DB8000_PART_STATUS".UNIT_02.STATION_1.PART_A.STATUS.PART_REJECTED )
      I_Contact( "DB8000_PART_STATUS".UNIT_02.STATION_1.PART_A.STATUS.UNIT_02_STATUS.FACE_R_STATION_3_DONE )
      I_Contact( "DB8000_PART_STATUS".UNIT_02.STATION_1.PART_A.STATUS.UNIT_02_STATUS.FACE_R_STATION_4_DONE )
   END_RUNG wire#w9
   RUNG wire#w11
      Contact( "DB4000_FIX_TABLE_POSITIONS".UNIT_02.FIXTURE_3.IN_LOAD_UNLOAD_STATION_1 )
   END_RUNG wire#w12
   RUNG wire#w11
      Contact( "DB4000_FIX_TABLE_POSITIONS".UNIT_02.FIXTURE_2.IN_LOAD_UNLOAD_STATION_1 )
      wire#w13
      I_Contact( "DB8000_PART_STATUS".UNIT_02.STATION_1.PART_A.STATUS.PART_REJECTED )
      I_Contact( "DB8000_PART_STATUS".UNIT_02.STATION_1.PART_A.STATUS.UNIT_02_STATUS.FACE_N_STATION_3_DONE )
      I_Contact( "DB8000_PART_STATUS".UNIT_02.STATION_1.PART_A.STATUS.UNIT_02_STATUS.FACE_N_STATION_4_DONE )
   END_RUNG wire#w9
   RUNG wire#w11
      Contact( "DB4000_FIX_TABLE_POSITIONS".UNIT_02.FIXTURE_4.IN_LOAD_UNLOAD_STATION_1 )
   END_RUNG wire#w13
   RUNG wire#powerrail
      Contact( "DB1101_MACHINE_SEQUENCE".SKIP_FIXTURE_UNIT_02 )
      Contact( "DB2430_FULL_DEPTH".FD_UNIT_02.FIX_IN_STA_1_FD )
      I_Contact( "DB8000_PART_STATUS".UNIT_02.STATION_1.PART_A.STATUS.PRESENT )
   END_RUNG wire#w9
   RUNG wire#powerrail
      Contact( "DB4000_FIX_TABLE_POSITIONS".UNIT_02.FIXTURE_1.IN_LOAD_UNLOAD_STATION_1 )
      wire#w14
      I_Contact( "DB7240_HARDWARE_SOFTWARE_ENABLE_DISABLE".DISABLE_FIXTURE.SW_UNIT_02_FIX_1_4_ENABLED )
   END_RUNG wire#w9
   RUNG wire#powerrail
      Contact( "DB4000_FIX_TABLE_POSITIONS".UNIT_02.FIXTURE_4.IN_LOAD_UNLOAD_STATION_1 )
   END_RUNG wire#w14
   RUNG wire#powerrail
      Contact( "DB4000_FIX_TABLE_POSITIONS".UNIT_02.FIXTURE_2.IN_LOAD_UNLOAD_STATION_1 )
      wire#w15
      I_Contact( "DB7240_HARDWARE_SOFTWARE_ENABLE_DISABLE".DISABLE_FIXTURE.SW_UNIT_02_FIX_2_3_ENABLED )
   END_RUNG wire#w9
   RUNG wire#powerrail
      Contact( "DB4000_FIX_TABLE_POSITIONS".UNIT_02.FIXTURE_3.IN_LOAD_UNLOAD_STATION_1 )
   END_RUNG wire#w15
   RUNG wire#powerrail
      Contact( "DB2031_CYCLES_GENERAL".CALIBRATION_CYCLE.CYCLE_SELECTED )
      I_Contact( "DB8000_PART_STATUS".UNIT_02.STATION_1.PART_A.STATUS.PRESENT )
      wire#w16
      Contact( "DB8000_PART_STATUS".UNIT_02.STATION_2.PART_A.STATUS.PRESENT )
   END_RUNG wire#w9
   RUNG wire#w16
      Contact( "DB8000_PART_STATUS".UNIT_02.STATION_3.PART_A.STATUS.PRESENT )
   END_RUNG wire#w9
   RUNG wire#w16
      Contact( "DB8000_PART_STATUS".UNIT_02.STATION_4.PART_A.STATUS.PRESENT )
   END_RUNG wire#w9
   // the same network as SCL:
   "DB1251_PART_CYCLE_UNIT_02".U02_STA_1_COND_OK_STA_0_CYCLE := (NOT "DB2031_CYCLES_GENERAL".RUN_OUT_UNIT_02.CYCLE_SELECTED AND (("DB2430_FULL_DEPTH".FD_UNIT_02.FIX_IN_STA_1_FD AND ((("DB4000_FIX_TABLE_POSITIONS".UNIT_02.FIXTURE_1.IN_LOAD_UNLOAD_STATION_1 OR "DB4000_FIX_TABLE_POSITIONS".UNIT_02.FIXTURE_3.IN_LOAD_UNLOAD_STATION_1) AND NOT "DB8000_PART_STATUS".UNIT_02.STATION_1.PART_A.STATUS.UNIT_02_STATUS.FACE_R_STATION_4_DONE) OR (("DB4000_FIX_TABLE_POSITIONS".UNIT_02.FIXTURE_2.IN_LOAD_UNLOAD_STATION_1 OR "DB4000_FIX_TABLE_POSITIONS".UNIT_02.FIXTURE_4.IN_LOAD_UNLOAD_STATION_1) AND NOT "DB8000_PART_STATUS".UNIT_02.STATION_1.PART_A.STATUS.UNIT_02_STATUS.FACE_N_STATION_4_DONE))) OR ("DB8000_PART_STATUS".UNIT_02.STATION_1.PART_A.STATUS.UNIT_02_STATUS.FACE_R_STATION_1_DONE AND NOT "DB8000_PART_STATUS".UNIT_02.STATION_1.PART_A.STATUS.PART_REJECTED AND NOT "DB8000_PART_STATUS".UNIT_02.STATION_1.PART_A.STATUS.UNIT_02_STATUS.FACE_R_STATION_3_DONE AND NOT "DB8000_PART_STATUS".UNIT_02.STATION_1.PART_A.STATUS.UNIT_02_STATUS.FACE_R_STATION_4_DONE AND ("DB4000_FIX_TABLE_POSITIONS".UNIT_02.FIXTURE_1.IN_LOAD_UNLOAD_STATION_1 OR "DB4000_FIX_TABLE_POSITIONS".UNIT_02.FIXTURE_3.IN_LOAD_UNLOAD_STATION_1)) OR ("DB8000_PART_STATUS".UNIT_02.STATION_1.PART_A.STATUS.UNIT_02_STATUS.FACE_N_STATION_1_DONE AND NOT "DB8000_PART_STATUS".UNIT_02.STATION_1.PART_A.STATUS.PART_REJECTED AND NOT "DB8000_PART_STATUS".UNIT_02.STATION_1.PART_A.STATUS.UNIT_02_STATUS.FACE_N_STATION_3_DONE AND NOT "DB8000_PART_STATUS".UNIT_02.STATION_1.PART_A.STATUS.UNIT_02_STATUS.FACE_N_STATION_4_DONE AND ("DB4000_FIX_TABLE_POSITIONS".UNIT_02.FIXTURE_2.IN_LOAD_UNLOAD_STATION_1 OR "DB4000_FIX_TABLE_POSITIONS".UNIT_02.FIXTURE_4.IN_LOAD_UNLOAD_STATION_1))) AND (("DB8000_PART_STATUS".UNIT_02.STATION_1.PART_A.STATUS.PRESENT AND NOT "DB8000_PART_STATUS".UNIT_02.STATION_1.PART_A.STATUS.VIRTUAL_PART AND (("DB4000_FIX_TABLE_POSITIONS".UNIT_02.FIXTURE_1.IN_LOAD_UNLOAD_STATION_1 AND "DB3500_UNIT_02_FIXTURE_1".CLAMPED_WITH_PART_ANALOG) OR ("DB4000_FIX_TABLE_POSITIONS".UNIT_02.FIXTURE_2.IN_LOAD_UNLOAD_STATION_1 AND "DB3600_UNIT_02_FIXTURE_2".CLAMPED_WITH_PART_ANALOG) OR ("DB4000_FIX_TABLE_POSITIONS".UNIT_02.FIXTURE_3.IN_LOAD_UNLOAD_STATION_1 AND "DB3700_UNIT_02_FIXTURE_3".CLAMPED_WITH_PART_ANALOG) OR ("DB4000_FIX_TABLE_POSITIONS".UNIT_02.FIXTURE_4.IN_LOAD_UNLOAD_STATION_1 AND "DB3800_UNIT_02_FIXTURE_4".CLAMPED_WITH_PART_ANALOG))) OR "DB8000_PART_STATUS".UNIT_02.STATION_1.PART_A.STATUS.VIRTUAL_PART)) OR ("DB2031_CYCLES_GENERAL".RUN_OUT_UNIT_02.CYCLE_SELECTED AND (NOT "DB8000_PART_STATUS".UNIT_02.STATION_1.PART_A.STATUS.PRESENT OR ("DB8000_PART_STATUS".UNIT_02.STATION_1.PART_A.STATUS.PRESENT AND ((("DB4000_FIX_TABLE_POSITIONS".UNIT_02.FIXTURE_1.IN_LOAD_UNLOAD_STATION_1 OR "DB4000_FIX_TABLE_POSITIONS".UNIT_02.FIXTURE_3.IN_LOAD_UNLOAD_STATION_1) AND NOT "DB8000_PART_STATUS".UNIT_02.STATION_1.PART_A.STATUS.PART_REJECTED AND NOT "DB8000_PART_STATUS".UNIT_02.STATION_1.PART_A.STATUS.UNIT_02_STATUS.FACE_R_STATION_3_DONE AND NOT "DB8000_PART_STATUS".UNIT_02.STATION_1.PART_A.STATUS.UNIT_02_STATUS.FACE_R_STATION_4_DONE) OR (("DB4000_FIX_TABLE_POSITIONS".UNIT_02.FIXTURE_2.IN_LOAD_UNLOAD_STATION_1 OR "DB4000_FIX_TABLE_POSITIONS".UNIT_02.FIXTURE_4.IN_LOAD_UNLOAD_STATION_1) AND NOT "DB8000_PART_STATUS".UNIT_02.STATION_1.PART_A.STATUS.PART_REJECTED AND NOT "DB8000_PART_STATUS".UNIT_02.STATION_1.PART_A.STATUS.UNIT_02_STATUS.FACE_N_STATION_3_DONE AND NOT "DB8000_PART_STATUS".UNIT_02.STATION_1.PART_A.STATUS.UNIT_02_STATUS.FACE_N_STATION_4_DONE))))) OR ("DB1101_MACHINE_SEQUENCE".SKIP_FIXTURE_UNIT_02 AND "DB2430_FULL_DEPTH".FD_UNIT_02.FIX_IN_STA_1_FD AND NOT "DB8000_PART_STATUS".UNIT_02.STATION_1.PART_A.STATUS.PRESENT) OR (("DB4000_FIX_TABLE_POSITIONS".UNIT_02.FIXTURE_1.IN_LOAD_UNLOAD_STATION_1 OR "DB4000_FIX_TABLE_POSITIONS".UNIT_02.FIXTURE_4.IN_LOAD_UNLOAD_STATION_1) AND NOT "DB7240_HARDWARE_SOFTWARE_ENABLE_DISABLE".DISABLE_FIXTURE.SW_UNIT_02_FIX_1_4_ENABLED) OR (("DB4000_FIX_TABLE_POSITIONS".UNIT_02.FIXTURE_2.IN_LOAD_UNLOAD_STATION_1 OR "DB4000_FIX_TABLE_POSITIONS".UNIT_02.FIXTURE_3.IN_LOAD_UNLOAD_STATION_1) AND NOT "DB7240_HARDWARE_SOFTWARE_ENABLE_DISABLE".DISABLE_FIXTURE.SW_UNIT_02_FIX_2_3_ENABLED) OR ("DB2031_CYCLES_GENERAL".CALIBRATION_CYCLE.CYCLE_SELECTED AND NOT "DB8000_PART_STATUS".UNIT_02.STATION_1.PART_A.STATUS.PRESENT AND ("DB8000_PART_STATUS".UNIT_02.STATION_2.PART_A.STATUS.PRESENT OR "DB8000_PART_STATUS".UNIT_02.STATION_3.PART_A.STATUS.PRESENT OR "DB8000_PART_STATUS".UNIT_02.STATION_4.PART_A.STATUS.PRESENT));
END_REGION

REGION Network 13: UNIT 02 STATION 2 CONDITIONS OK FOR STATION 0 CYCLE REQUEST
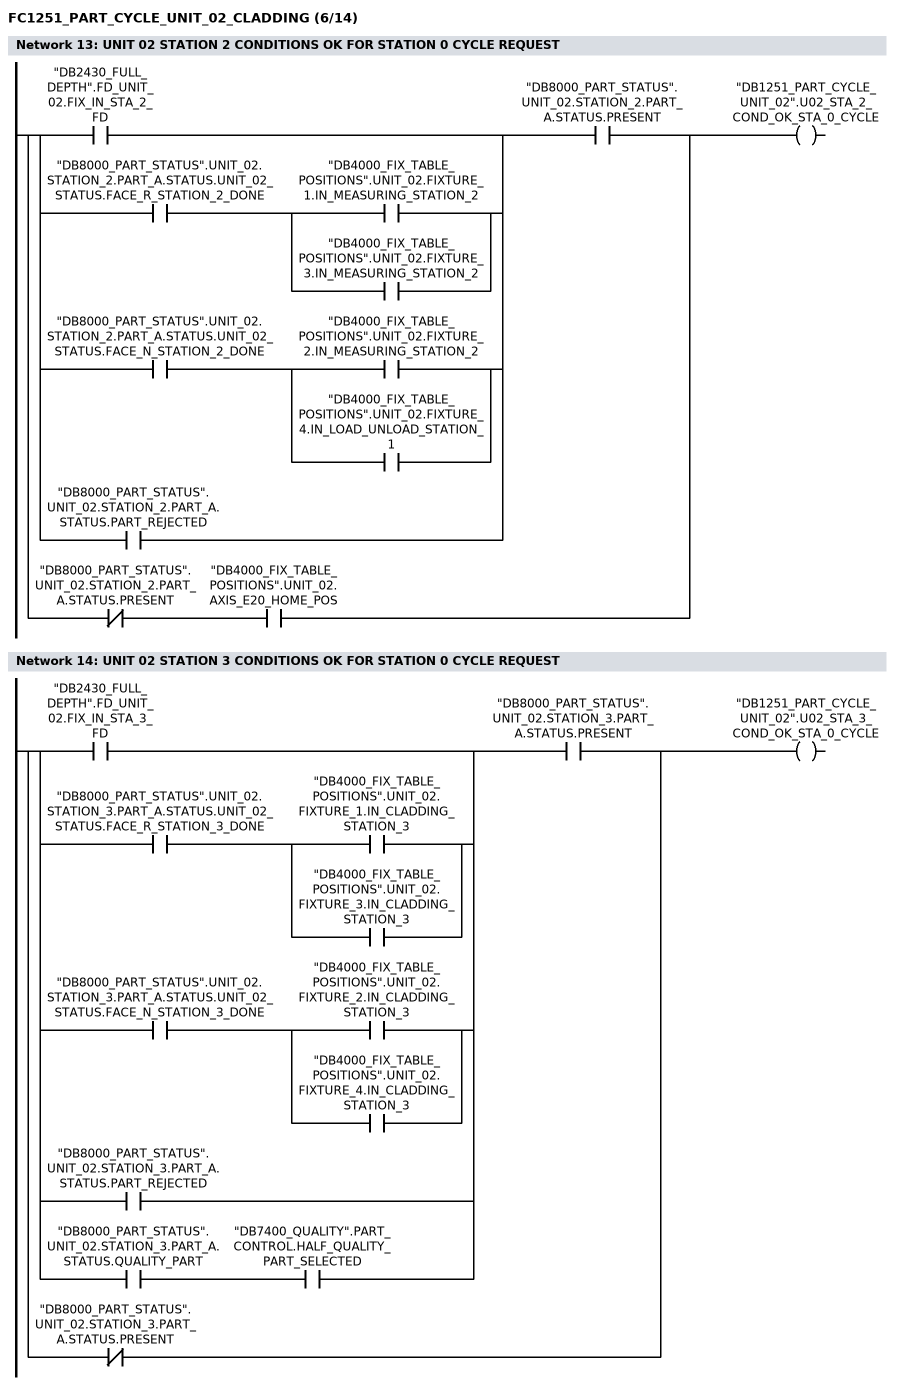
   RUNG wire#powerrail
      Contact( "DB2430_FULL_DEPTH".FD_UNIT_02.FIX_IN_STA_2_FD )
      wire#w1
      Contact( "DB8000_PART_STATUS".UNIT_02.STATION_2.PART_A.STATUS.PRESENT )
      wire#w4
      Coil( "DB1251_PART_CYCLE_UNIT_02".U02_STA_2_COND_OK_STA_0_CYCLE )
   END_RUNG
   RUNG wire#powerrail
      Contact( "DB8000_PART_STATUS".UNIT_02.STATION_2.PART_A.STATUS.UNIT_02_STATUS.FACE_R_STATION_2_DONE )
      wire#w2
      Contact( "DB4000_FIX_TABLE_POSITIONS".UNIT_02.FIXTURE_1.IN_MEASURING_STATION_2 )
   END_RUNG wire#w1
   RUNG wire#w2
      Contact( "DB4000_FIX_TABLE_POSITIONS".UNIT_02.FIXTURE_3.IN_MEASURING_STATION_2 )
   END_RUNG wire#w1
   RUNG wire#powerrail
      Contact( "DB8000_PART_STATUS".UNIT_02.STATION_2.PART_A.STATUS.UNIT_02_STATUS.FACE_N_STATION_2_DONE )
      wire#w3
      Contact( "DB4000_FIX_TABLE_POSITIONS".UNIT_02.FIXTURE_2.IN_MEASURING_STATION_2 )
   END_RUNG wire#w1
   RUNG wire#w3
      Contact( "DB4000_FIX_TABLE_POSITIONS".UNIT_02.FIXTURE_4.IN_LOAD_UNLOAD_STATION_1 )
   END_RUNG wire#w1
   RUNG wire#powerrail
      Contact( "DB8000_PART_STATUS".UNIT_02.STATION_2.PART_A.STATUS.PART_REJECTED )
   END_RUNG wire#w1
   RUNG wire#powerrail
      I_Contact( "DB8000_PART_STATUS".UNIT_02.STATION_2.PART_A.STATUS.PRESENT )
      Contact( "DB4000_FIX_TABLE_POSITIONS".UNIT_02.AXIS_E20_HOME_POS )
   END_RUNG wire#w4
   // the same network as SCL:
   "DB1251_PART_CYCLE_UNIT_02".U02_STA_2_COND_OK_STA_0_CYCLE := (("DB2430_FULL_DEPTH".FD_UNIT_02.FIX_IN_STA_2_FD OR ("DB8000_PART_STATUS".UNIT_02.STATION_2.PART_A.STATUS.UNIT_02_STATUS.FACE_R_STATION_2_DONE AND ("DB4000_FIX_TABLE_POSITIONS".UNIT_02.FIXTURE_1.IN_MEASURING_STATION_2 OR "DB4000_FIX_TABLE_POSITIONS".UNIT_02.FIXTURE_3.IN_MEASURING_STATION_2)) OR ("DB8000_PART_STATUS".UNIT_02.STATION_2.PART_A.STATUS.UNIT_02_STATUS.FACE_N_STATION_2_DONE AND ("DB4000_FIX_TABLE_POSITIONS".UNIT_02.FIXTURE_2.IN_MEASURING_STATION_2 OR "DB4000_FIX_TABLE_POSITIONS".UNIT_02.FIXTURE_4.IN_LOAD_UNLOAD_STATION_1)) OR "DB8000_PART_STATUS".UNIT_02.STATION_2.PART_A.STATUS.PART_REJECTED) AND "DB8000_PART_STATUS".UNIT_02.STATION_2.PART_A.STATUS.PRESENT) OR (NOT "DB8000_PART_STATUS".UNIT_02.STATION_2.PART_A.STATUS.PRESENT AND "DB4000_FIX_TABLE_POSITIONS".UNIT_02.AXIS_E20_HOME_POS);
END_REGION

REGION Network 14: UNIT 02 STATION 3 CONDITIONS OK FOR STATION 0 CYCLE REQUEST
   RUNG wire#powerrail
      Contact( "DB2430_FULL_DEPTH".FD_UNIT_02.FIX_IN_STA_3_FD )
      wire#w1
      Contact( "DB8000_PART_STATUS".UNIT_02.STATION_3.PART_A.STATUS.PRESENT )
      wire#w4
      Coil( "DB1251_PART_CYCLE_UNIT_02".U02_STA_3_COND_OK_STA_0_CYCLE )
   END_RUNG
   RUNG wire#powerrail
      Contact( "DB8000_PART_STATUS".UNIT_02.STATION_3.PART_A.STATUS.UNIT_02_STATUS.FACE_R_STATION_3_DONE )
      wire#w2
      Contact( "DB4000_FIX_TABLE_POSITIONS".UNIT_02.FIXTURE_1.IN_CLADDING_STATION_3 )
   END_RUNG wire#w1
   RUNG wire#w2
      Contact( "DB4000_FIX_TABLE_POSITIONS".UNIT_02.FIXTURE_3.IN_CLADDING_STATION_3 )
   END_RUNG wire#w1
   RUNG wire#powerrail
      Contact( "DB8000_PART_STATUS".UNIT_02.STATION_3.PART_A.STATUS.UNIT_02_STATUS.FACE_N_STATION_3_DONE )
      wire#w3
      Contact( "DB4000_FIX_TABLE_POSITIONS".UNIT_02.FIXTURE_2.IN_CLADDING_STATION_3 )
   END_RUNG wire#w1
   RUNG wire#w3
      Contact( "DB4000_FIX_TABLE_POSITIONS".UNIT_02.FIXTURE_4.IN_CLADDING_STATION_3 )
   END_RUNG wire#w1
   RUNG wire#powerrail
      Contact( "DB8000_PART_STATUS".UNIT_02.STATION_3.PART_A.STATUS.PART_REJECTED )
   END_RUNG wire#w1
   RUNG wire#powerrail
      Contact( "DB8000_PART_STATUS".UNIT_02.STATION_3.PART_A.STATUS.QUALITY_PART )
      Contact( "DB7400_QUALITY".PART_CONTROL.HALF_QUALITY_PART_SELECTED )
   END_RUNG wire#w1
   RUNG wire#powerrail
      I_Contact( "DB8000_PART_STATUS".UNIT_02.STATION_3.PART_A.STATUS.PRESENT )
   END_RUNG wire#w4
   // the same network as SCL:
   "DB1251_PART_CYCLE_UNIT_02".U02_STA_3_COND_OK_STA_0_CYCLE := (("DB2430_FULL_DEPTH".FD_UNIT_02.FIX_IN_STA_3_FD OR ("DB8000_PART_STATUS".UNIT_02.STATION_3.PART_A.STATUS.UNIT_02_STATUS.FACE_R_STATION_3_DONE AND ("DB4000_FIX_TABLE_POSITIONS".UNIT_02.FIXTURE_1.IN_CLADDING_STATION_3 OR "DB4000_FIX_TABLE_POSITIONS".UNIT_02.FIXTURE_3.IN_CLADDING_STATION_3)) OR ("DB8000_PART_STATUS".UNIT_02.STATION_3.PART_A.STATUS.UNIT_02_STATUS.FACE_N_STATION_3_DONE AND ("DB4000_FIX_TABLE_POSITIONS".UNIT_02.FIXTURE_2.IN_CLADDING_STATION_3 OR "DB4000_FIX_TABLE_POSITIONS".UNIT_02.FIXTURE_4.IN_CLADDING_STATION_3)) OR "DB8000_PART_STATUS".UNIT_02.STATION_3.PART_A.STATUS.PART_REJECTED OR ("DB8000_PART_STATUS".UNIT_02.STATION_3.PART_A.STATUS.QUALITY_PART AND "DB7400_QUALITY".PART_CONTROL.HALF_QUALITY_PART_SELECTED)) AND "DB8000_PART_STATUS".UNIT_02.STATION_3.PART_A.STATUS.PRESENT) OR NOT "DB8000_PART_STATUS".UNIT_02.STATION_3.PART_A.STATUS.PRESENT;
END_REGION

REGION Network 15: UNIT 02 STATION 4 CONDITIONS OK FOR STATION 0 CYCLE REQUEST
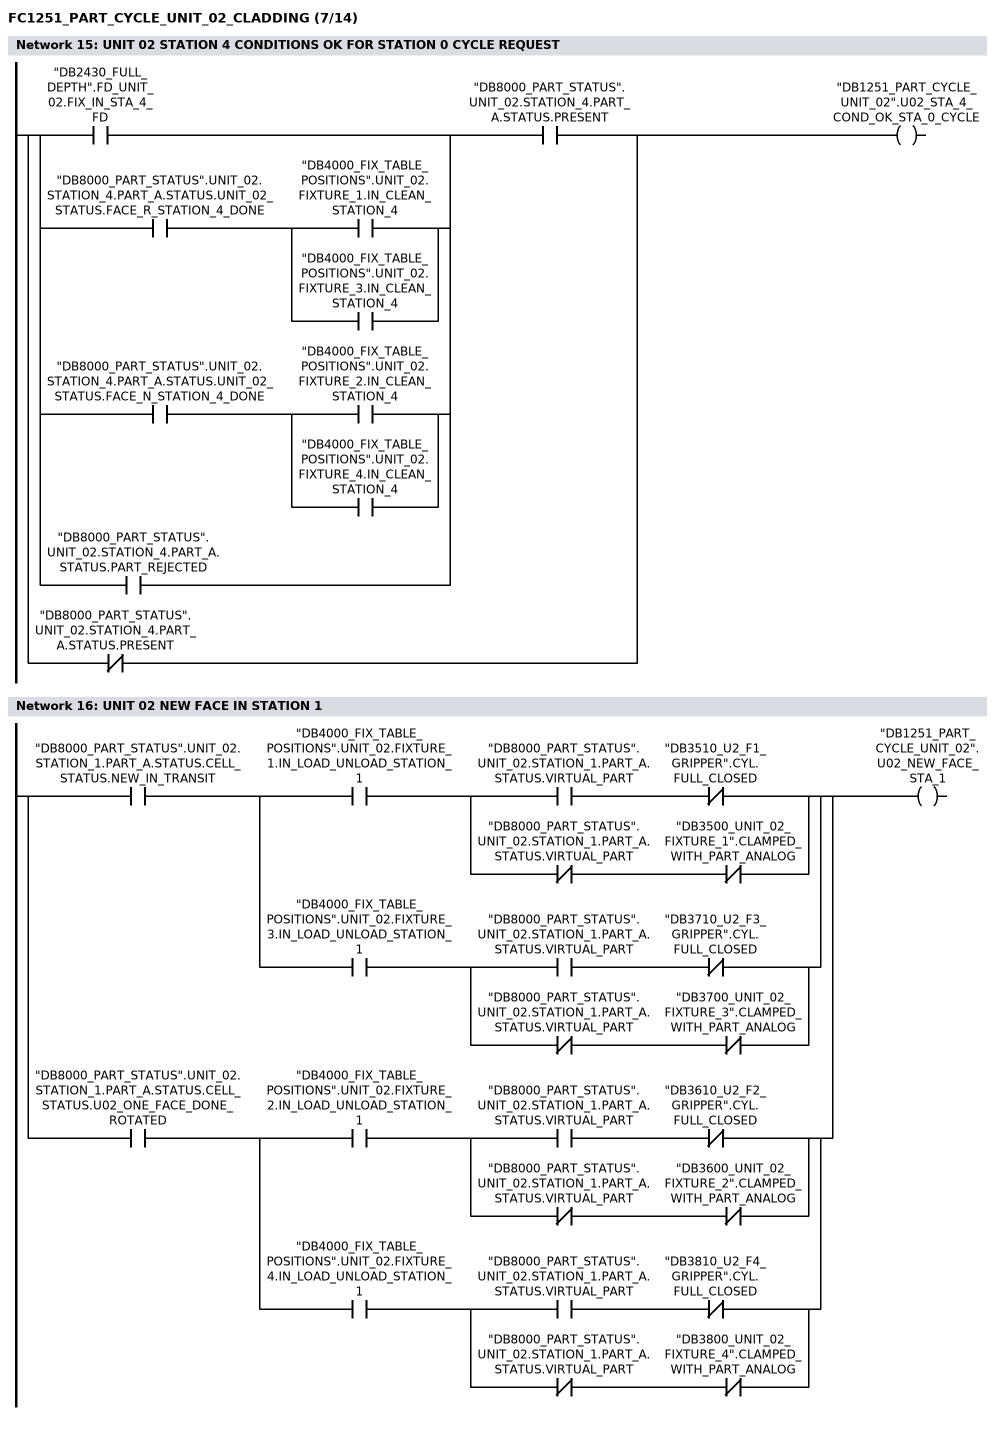
   RUNG wire#powerrail
      Contact( "DB2430_FULL_DEPTH".FD_UNIT_02.FIX_IN_STA_4_FD )
      wire#w1
      Contact( "DB8000_PART_STATUS".UNIT_02.STATION_4.PART_A.STATUS.PRESENT )
      wire#w4
      Coil( "DB1251_PART_CYCLE_UNIT_02".U02_STA_4_COND_OK_STA_0_CYCLE )
   END_RUNG
   RUNG wire#powerrail
      Contact( "DB8000_PART_STATUS".UNIT_02.STATION_4.PART_A.STATUS.UNIT_02_STATUS.FACE_R_STATION_4_DONE )
      wire#w2
      Contact( "DB4000_FIX_TABLE_POSITIONS".UNIT_02.FIXTURE_1.IN_CLEAN_STATION_4 )
   END_RUNG wire#w1
   RUNG wire#w2
      Contact( "DB4000_FIX_TABLE_POSITIONS".UNIT_02.FIXTURE_3.IN_CLEAN_STATION_4 )
   END_RUNG wire#w1
   RUNG wire#powerrail
      Contact( "DB8000_PART_STATUS".UNIT_02.STATION_4.PART_A.STATUS.UNIT_02_STATUS.FACE_N_STATION_4_DONE )
      wire#w3
      Contact( "DB4000_FIX_TABLE_POSITIONS".UNIT_02.FIXTURE_2.IN_CLEAN_STATION_4 )
   END_RUNG wire#w1
   RUNG wire#w3
      Contact( "DB4000_FIX_TABLE_POSITIONS".UNIT_02.FIXTURE_4.IN_CLEAN_STATION_4 )
   END_RUNG wire#w1
   RUNG wire#powerrail
      Contact( "DB8000_PART_STATUS".UNIT_02.STATION_4.PART_A.STATUS.PART_REJECTED )
   END_RUNG wire#w1
   RUNG wire#powerrail
      I_Contact( "DB8000_PART_STATUS".UNIT_02.STATION_4.PART_A.STATUS.PRESENT )
   END_RUNG wire#w4
   // the same network as SCL:
   "DB1251_PART_CYCLE_UNIT_02".U02_STA_4_COND_OK_STA_0_CYCLE := (("DB2430_FULL_DEPTH".FD_UNIT_02.FIX_IN_STA_4_FD OR ("DB8000_PART_STATUS".UNIT_02.STATION_4.PART_A.STATUS.UNIT_02_STATUS.FACE_R_STATION_4_DONE AND ("DB4000_FIX_TABLE_POSITIONS".UNIT_02.FIXTURE_1.IN_CLEAN_STATION_4 OR "DB4000_FIX_TABLE_POSITIONS".UNIT_02.FIXTURE_3.IN_CLEAN_STATION_4)) OR ("DB8000_PART_STATUS".UNIT_02.STATION_4.PART_A.STATUS.UNIT_02_STATUS.FACE_N_STATION_4_DONE AND ("DB4000_FIX_TABLE_POSITIONS".UNIT_02.FIXTURE_2.IN_CLEAN_STATION_4 OR "DB4000_FIX_TABLE_POSITIONS".UNIT_02.FIXTURE_4.IN_CLEAN_STATION_4)) OR "DB8000_PART_STATUS".UNIT_02.STATION_4.PART_A.STATUS.PART_REJECTED) AND "DB8000_PART_STATUS".UNIT_02.STATION_4.PART_A.STATUS.PRESENT) OR NOT "DB8000_PART_STATUS".UNIT_02.STATION_4.PART_A.STATUS.PRESENT;
END_REGION

REGION Network 16: UNIT 02 NEW FACE IN STATION 1
   RUNG wire#powerrail
      Contact( "DB8000_PART_STATUS".UNIT_02.STATION_1.PART_A.STATUS.CELL_STATUS.NEW_IN_TRANSIT )
      wire#w1
      Contact( "DB4000_FIX_TABLE_POSITIONS".UNIT_02.FIXTURE_1.IN_LOAD_UNLOAD_STATION_1 )
      wire#w2
      Contact( "DB8000_PART_STATUS".UNIT_02.STATION_1.PART_A.STATUS.VIRTUAL_PART )
      I_Contact( "DB3510_U2_F1_GRIPPER".CYL.FULL_CLOSED )
      wire#w3
      Coil( "DB1251_PART_CYCLE_UNIT_02".U02_NEW_FACE_STA_1 )
   END_RUNG
   RUNG wire#w2
      I_Contact( "DB8000_PART_STATUS".UNIT_02.STATION_1.PART_A.STATUS.VIRTUAL_PART )
      I_Contact( "DB3500_UNIT_02_FIXTURE_1".CLAMPED_WITH_PART_ANALOG )
   END_RUNG wire#w3
   RUNG wire#w1
      Contact( "DB4000_FIX_TABLE_POSITIONS".UNIT_02.FIXTURE_3.IN_LOAD_UNLOAD_STATION_1 )
      wire#w4
      Contact( "DB8000_PART_STATUS".UNIT_02.STATION_1.PART_A.STATUS.VIRTUAL_PART )
      I_Contact( "DB3710_U2_F3_GRIPPER".CYL.FULL_CLOSED )
   END_RUNG wire#w3
   RUNG wire#w4
      I_Contact( "DB8000_PART_STATUS".UNIT_02.STATION_1.PART_A.STATUS.VIRTUAL_PART )
      I_Contact( "DB3700_UNIT_02_FIXTURE_3".CLAMPED_WITH_PART_ANALOG )
   END_RUNG wire#w3
   RUNG wire#powerrail
      Contact( "DB8000_PART_STATUS".UNIT_02.STATION_1.PART_A.STATUS.CELL_STATUS.U02_ONE_FACE_DONE_ROTATED )
      wire#w5
      Contact( "DB4000_FIX_TABLE_POSITIONS".UNIT_02.FIXTURE_2.IN_LOAD_UNLOAD_STATION_1 )
      wire#w6
      Contact( "DB8000_PART_STATUS".UNIT_02.STATION_1.PART_A.STATUS.VIRTUAL_PART )
      I_Contact( "DB3610_U2_F2_GRIPPER".CYL.FULL_CLOSED )
   END_RUNG wire#w3
   RUNG wire#w6
      I_Contact( "DB8000_PART_STATUS".UNIT_02.STATION_1.PART_A.STATUS.VIRTUAL_PART )
      I_Contact( "DB3600_UNIT_02_FIXTURE_2".CLAMPED_WITH_PART_ANALOG )
   END_RUNG wire#w3
   RUNG wire#w5
      Contact( "DB4000_FIX_TABLE_POSITIONS".UNIT_02.FIXTURE_4.IN_LOAD_UNLOAD_STATION_1 )
      wire#w7
      Contact( "DB8000_PART_STATUS".UNIT_02.STATION_1.PART_A.STATUS.VIRTUAL_PART )
      I_Contact( "DB3810_U2_F4_GRIPPER".CYL.FULL_CLOSED )
   END_RUNG wire#w3
   RUNG wire#w7
      I_Contact( "DB8000_PART_STATUS".UNIT_02.STATION_1.PART_A.STATUS.VIRTUAL_PART )
      I_Contact( "DB3800_UNIT_02_FIXTURE_4".CLAMPED_WITH_PART_ANALOG )
   END_RUNG wire#w3
   // the same network as SCL:
   "DB1251_PART_CYCLE_UNIT_02".U02_NEW_FACE_STA_1 := ("DB8000_PART_STATUS".UNIT_02.STATION_1.PART_A.STATUS.CELL_STATUS.NEW_IN_TRANSIT AND (("DB4000_FIX_TABLE_POSITIONS".UNIT_02.FIXTURE_1.IN_LOAD_UNLOAD_STATION_1 AND (("DB8000_PART_STATUS".UNIT_02.STATION_1.PART_A.STATUS.VIRTUAL_PART AND NOT "DB3510_U2_F1_GRIPPER".CYL.FULL_CLOSED) OR (NOT "DB8000_PART_STATUS".UNIT_02.STATION_1.PART_A.STATUS.VIRTUAL_PART AND NOT "DB3500_UNIT_02_FIXTURE_1".CLAMPED_WITH_PART_ANALOG))) OR ("DB4000_FIX_TABLE_POSITIONS".UNIT_02.FIXTURE_3.IN_LOAD_UNLOAD_STATION_1 AND (("DB8000_PART_STATUS".UNIT_02.STATION_1.PART_A.STATUS.VIRTUAL_PART AND NOT "DB3710_U2_F3_GRIPPER".CYL.FULL_CLOSED) OR (NOT "DB8000_PART_STATUS".UNIT_02.STATION_1.PART_A.STATUS.VIRTUAL_PART AND NOT "DB3700_UNIT_02_FIXTURE_3".CLAMPED_WITH_PART_ANALOG))))) OR ("DB8000_PART_STATUS".UNIT_02.STATION_1.PART_A.STATUS.CELL_STATUS.U02_ONE_FACE_DONE_ROTATED AND (("DB4000_FIX_TABLE_POSITIONS".UNIT_02.FIXTURE_2.IN_LOAD_UNLOAD_STATION_1 AND (("DB8000_PART_STATUS".UNIT_02.STATION_1.PART_A.STATUS.VIRTUAL_PART AND NOT "DB3610_U2_F2_GRIPPER".CYL.FULL_CLOSED) OR (NOT "DB8000_PART_STATUS".UNIT_02.STATION_1.PART_A.STATUS.VIRTUAL_PART AND NOT "DB3600_UNIT_02_FIXTURE_2".CLAMPED_WITH_PART_ANALOG))) OR ("DB4000_FIX_TABLE_POSITIONS".UNIT_02.FIXTURE_4.IN_LOAD_UNLOAD_STATION_1 AND (("DB8000_PART_STATUS".UNIT_02.STATION_1.PART_A.STATUS.VIRTUAL_PART AND NOT "DB3810_U2_F4_GRIPPER".CYL.FULL_CLOSED) OR (NOT "DB8000_PART_STATUS".UNIT_02.STATION_1.PART_A.STATUS.VIRTUAL_PART AND NOT "DB3800_UNIT_02_FIXTURE_4".CLAMPED_WITH_PART_ANALOG)))));
END_REGION

REGION Network 17: UNIT 02 FACE DONE IN STATION 1
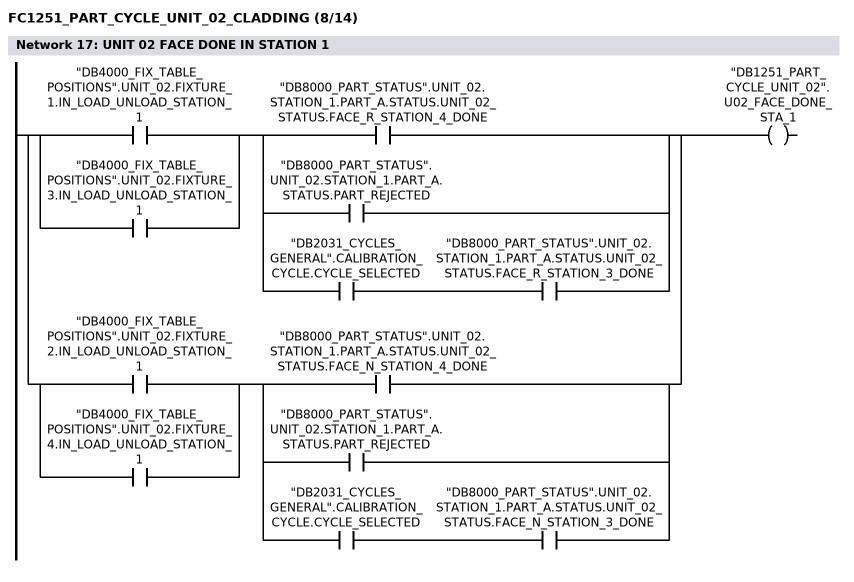
   RUNG wire#powerrail
      Contact( "DB4000_FIX_TABLE_POSITIONS".UNIT_02.FIXTURE_1.IN_LOAD_UNLOAD_STATION_1 )
      wire#w1
      Contact( "DB8000_PART_STATUS".UNIT_02.STATION_1.PART_A.STATUS.UNIT_02_STATUS.FACE_R_STATION_4_DONE )
      wire#w2
      Coil( "DB1251_PART_CYCLE_UNIT_02".U02_FACE_DONE_STA_1 )
   END_RUNG
   RUNG wire#powerrail
      Contact( "DB4000_FIX_TABLE_POSITIONS".UNIT_02.FIXTURE_3.IN_LOAD_UNLOAD_STATION_1 )
   END_RUNG wire#w1
   RUNG wire#w1
      Contact( "DB8000_PART_STATUS".UNIT_02.STATION_1.PART_A.STATUS.PART_REJECTED )
   END_RUNG wire#w2
   RUNG wire#w1
      Contact( "DB2031_CYCLES_GENERAL".CALIBRATION_CYCLE.CYCLE_SELECTED )
      Contact( "DB8000_PART_STATUS".UNIT_02.STATION_1.PART_A.STATUS.UNIT_02_STATUS.FACE_R_STATION_3_DONE )
   END_RUNG wire#w2
   RUNG wire#powerrail
      Contact( "DB4000_FIX_TABLE_POSITIONS".UNIT_02.FIXTURE_2.IN_LOAD_UNLOAD_STATION_1 )
      wire#w3
      Contact( "DB8000_PART_STATUS".UNIT_02.STATION_1.PART_A.STATUS.UNIT_02_STATUS.FACE_N_STATION_4_DONE )
   END_RUNG wire#w2
   RUNG wire#powerrail
      Contact( "DB4000_FIX_TABLE_POSITIONS".UNIT_02.FIXTURE_4.IN_LOAD_UNLOAD_STATION_1 )
   END_RUNG wire#w3
   RUNG wire#w3
      Contact( "DB8000_PART_STATUS".UNIT_02.STATION_1.PART_A.STATUS.PART_REJECTED )
   END_RUNG wire#w2
   RUNG wire#w3
      Contact( "DB2031_CYCLES_GENERAL".CALIBRATION_CYCLE.CYCLE_SELECTED )
      Contact( "DB8000_PART_STATUS".UNIT_02.STATION_1.PART_A.STATUS.UNIT_02_STATUS.FACE_N_STATION_3_DONE )
   END_RUNG wire#w2
   // the same network as SCL:
   "DB1251_PART_CYCLE_UNIT_02".U02_FACE_DONE_STA_1 := (("DB4000_FIX_TABLE_POSITIONS".UNIT_02.FIXTURE_1.IN_LOAD_UNLOAD_STATION_1 OR "DB4000_FIX_TABLE_POSITIONS".UNIT_02.FIXTURE_3.IN_LOAD_UNLOAD_STATION_1) AND ("DB8000_PART_STATUS".UNIT_02.STATION_1.PART_A.STATUS.UNIT_02_STATUS.FACE_R_STATION_4_DONE OR "DB8000_PART_STATUS".UNIT_02.STATION_1.PART_A.STATUS.PART_REJECTED OR ("DB2031_CYCLES_GENERAL".CALIBRATION_CYCLE.CYCLE_SELECTED AND "DB8000_PART_STATUS".UNIT_02.STATION_1.PART_A.STATUS.UNIT_02_STATUS.FACE_R_STATION_3_DONE))) OR (("DB4000_FIX_TABLE_POSITIONS".UNIT_02.FIXTURE_2.IN_LOAD_UNLOAD_STATION_1 OR "DB4000_FIX_TABLE_POSITIONS".UNIT_02.FIXTURE_4.IN_LOAD_UNLOAD_STATION_1) AND ("DB8000_PART_STATUS".UNIT_02.STATION_1.PART_A.STATUS.UNIT_02_STATUS.FACE_N_STATION_4_DONE OR "DB8000_PART_STATUS".UNIT_02.STATION_1.PART_A.STATUS.PART_REJECTED OR ("DB2031_CYCLES_GENERAL".CALIBRATION_CYCLE.CYCLE_SELECTED AND "DB8000_PART_STATUS".UNIT_02.STATION_1.PART_A.STATUS.UNIT_02_STATUS.FACE_N_STATION_3_DONE)));
END_REGION

REGION Network 18: CYCLE UNIT 02 STATION 0
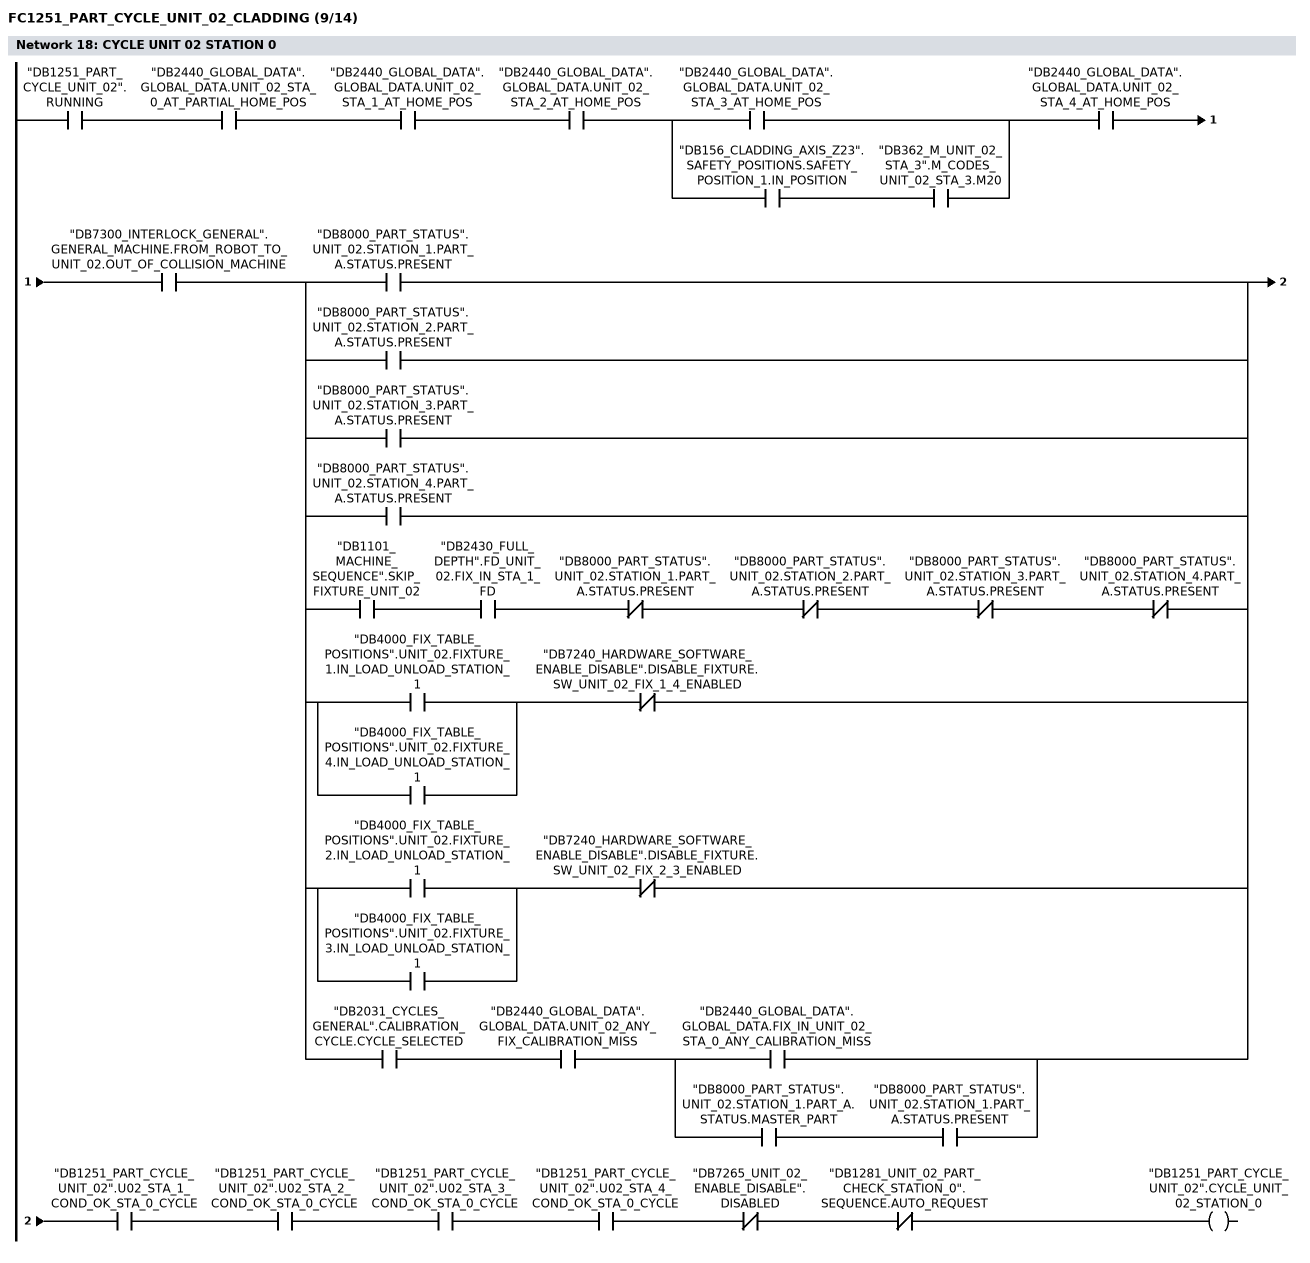
   RUNG wire#powerrail
      Contact( "DB1251_PART_CYCLE_UNIT_02".RUNNING )
      Contact( "DB2440_GLOBAL_DATA".GLOBAL_DATA.UNIT_02_STA_0_AT_PARTIAL_HOME_POS )
      Contact( "DB2440_GLOBAL_DATA".GLOBAL_DATA.UNIT_02_STA_1_AT_HOME_POS )
      Contact( "DB2440_GLOBAL_DATA".GLOBAL_DATA.UNIT_02_STA_2_AT_HOME_POS )
      wire#w1
      Contact( "DB2440_GLOBAL_DATA".GLOBAL_DATA.UNIT_02_STA_3_AT_HOME_POS )
      wire#w2
      Contact( "DB2440_GLOBAL_DATA".GLOBAL_DATA.UNIT_02_STA_4_AT_HOME_POS )
      Contact( "DB7300_INTERLOCK_GENERAL".GENERAL_MACHINE.FROM_ROBOT_TO_UNIT_02.OUT_OF_COLLISION_MACHINE )
      wire#w3
      Contact( "DB8000_PART_STATUS".UNIT_02.STATION_1.PART_A.STATUS.PRESENT )
      wire#w4
      Contact( "DB1251_PART_CYCLE_UNIT_02".U02_STA_1_COND_OK_STA_0_CYCLE )
      Contact( "DB1251_PART_CYCLE_UNIT_02".U02_STA_2_COND_OK_STA_0_CYCLE )
      Contact( "DB1251_PART_CYCLE_UNIT_02".U02_STA_3_COND_OK_STA_0_CYCLE )
      Contact( "DB1251_PART_CYCLE_UNIT_02".U02_STA_4_COND_OK_STA_0_CYCLE )
      I_Contact( "DB7265_UNIT_02_ENABLE_DISABLE".DISABLED )
      I_Contact( "DB1281_UNIT_02_PART_CHECK_STATION_0".SEQUENCE.AUTO_REQUEST )
      Coil( "DB1251_PART_CYCLE_UNIT_02".CYCLE_UNIT_02_STATION_0 )
   END_RUNG
   RUNG wire#w1
      Contact( "DB156_CLADDING_AXIS_Z23".SAFETY_POSITIONS.SAFETY_POSITION_1.IN_POSITION )
      Contact( "DB362_M_UNIT_02_STA_3".M_CODES_UNIT_02_STA_3.M20 )
   END_RUNG wire#w2
   RUNG wire#w3
      Contact( "DB8000_PART_STATUS".UNIT_02.STATION_2.PART_A.STATUS.PRESENT )
   END_RUNG wire#w4
   RUNG wire#w3
      Contact( "DB8000_PART_STATUS".UNIT_02.STATION_3.PART_A.STATUS.PRESENT )
   END_RUNG wire#w4
   RUNG wire#w3
      Contact( "DB8000_PART_STATUS".UNIT_02.STATION_4.PART_A.STATUS.PRESENT )
   END_RUNG wire#w4
   RUNG wire#w3
      Contact( "DB1101_MACHINE_SEQUENCE".SKIP_FIXTURE_UNIT_02 )
      Contact( "DB2430_FULL_DEPTH".FD_UNIT_02.FIX_IN_STA_1_FD )
      I_Contact( "DB8000_PART_STATUS".UNIT_02.STATION_1.PART_A.STATUS.PRESENT )
      I_Contact( "DB8000_PART_STATUS".UNIT_02.STATION_2.PART_A.STATUS.PRESENT )
      I_Contact( "DB8000_PART_STATUS".UNIT_02.STATION_3.PART_A.STATUS.PRESENT )
      I_Contact( "DB8000_PART_STATUS".UNIT_02.STATION_4.PART_A.STATUS.PRESENT )
   END_RUNG wire#w4
   RUNG wire#w3
      Contact( "DB4000_FIX_TABLE_POSITIONS".UNIT_02.FIXTURE_1.IN_LOAD_UNLOAD_STATION_1 )
      wire#w5
      I_Contact( "DB7240_HARDWARE_SOFTWARE_ENABLE_DISABLE".DISABLE_FIXTURE.SW_UNIT_02_FIX_1_4_ENABLED )
   END_RUNG wire#w4
   RUNG wire#w3
      Contact( "DB4000_FIX_TABLE_POSITIONS".UNIT_02.FIXTURE_4.IN_LOAD_UNLOAD_STATION_1 )
   END_RUNG wire#w5
   RUNG wire#w3
      Contact( "DB4000_FIX_TABLE_POSITIONS".UNIT_02.FIXTURE_2.IN_LOAD_UNLOAD_STATION_1 )
      wire#w6
      I_Contact( "DB7240_HARDWARE_SOFTWARE_ENABLE_DISABLE".DISABLE_FIXTURE.SW_UNIT_02_FIX_2_3_ENABLED )
   END_RUNG wire#w4
   RUNG wire#w3
      Contact( "DB4000_FIX_TABLE_POSITIONS".UNIT_02.FIXTURE_3.IN_LOAD_UNLOAD_STATION_1 )
   END_RUNG wire#w6
   RUNG wire#w3
      Contact( "DB2031_CYCLES_GENERAL".CALIBRATION_CYCLE.CYCLE_SELECTED )
      Contact( "DB2440_GLOBAL_DATA".GLOBAL_DATA.UNIT_02_ANY_FIX_CALIBRATION_MISS )
      wire#w7
      Contact( "DB2440_GLOBAL_DATA".GLOBAL_DATA.FIX_IN_UNIT_02_STA_0_ANY_CALIBRATION_MISS )
   END_RUNG wire#w4
   RUNG wire#w7
      Contact( "DB8000_PART_STATUS".UNIT_02.STATION_1.PART_A.STATUS.MASTER_PART )
      Contact( "DB8000_PART_STATUS".UNIT_02.STATION_1.PART_A.STATUS.PRESENT )
   END_RUNG wire#w4
   // the same network as SCL:
   "DB1251_PART_CYCLE_UNIT_02".CYCLE_UNIT_02_STATION_0 := "DB1251_PART_CYCLE_UNIT_02".RUNNING AND "DB2440_GLOBAL_DATA".GLOBAL_DATA.UNIT_02_STA_0_AT_PARTIAL_HOME_POS AND "DB2440_GLOBAL_DATA".GLOBAL_DATA.UNIT_02_STA_1_AT_HOME_POS AND "DB2440_GLOBAL_DATA".GLOBAL_DATA.UNIT_02_STA_2_AT_HOME_POS AND ("DB2440_GLOBAL_DATA".GLOBAL_DATA.UNIT_02_STA_3_AT_HOME_POS OR ("DB156_CLADDING_AXIS_Z23".SAFETY_POSITIONS.SAFETY_POSITION_1.IN_POSITION AND "DB362_M_UNIT_02_STA_3".M_CODES_UNIT_02_STA_3.M20)) AND "DB2440_GLOBAL_DATA".GLOBAL_DATA.UNIT_02_STA_4_AT_HOME_POS AND "DB7300_INTERLOCK_GENERAL".GENERAL_MACHINE.FROM_ROBOT_TO_UNIT_02.OUT_OF_COLLISION_MACHINE AND ("DB8000_PART_STATUS".UNIT_02.STATION_1.PART_A.STATUS.PRESENT OR "DB8000_PART_STATUS".UNIT_02.STATION_2.PART_A.STATUS.PRESENT OR "DB8000_PART_STATUS".UNIT_02.STATION_3.PART_A.STATUS.PRESENT OR "DB8000_PART_STATUS".UNIT_02.STATION_4.PART_A.STATUS.PRESENT OR ("DB1101_MACHINE_SEQUENCE".SKIP_FIXTURE_UNIT_02 AND "DB2430_FULL_DEPTH".FD_UNIT_02.FIX_IN_STA_1_FD AND NOT "DB8000_PART_STATUS".UNIT_02.STATION_1.PART_A.STATUS.PRESENT AND NOT "DB8000_PART_STATUS".UNIT_02.STATION_2.PART_A.STATUS.PRESENT AND NOT "DB8000_PART_STATUS".UNIT_02.STATION_3.PART_A.STATUS.PRESENT AND NOT "DB8000_PART_STATUS".UNIT_02.STATION_4.PART_A.STATUS.PRESENT) OR (("DB4000_FIX_TABLE_POSITIONS".UNIT_02.FIXTURE_1.IN_LOAD_UNLOAD_STATION_1 OR "DB4000_FIX_TABLE_POSITIONS".UNIT_02.FIXTURE_4.IN_LOAD_UNLOAD_STATION_1) AND NOT "DB7240_HARDWARE_SOFTWARE_ENABLE_DISABLE".DISABLE_FIXTURE.SW_UNIT_02_FIX_1_4_ENABLED) OR (("DB4000_FIX_TABLE_POSITIONS".UNIT_02.FIXTURE_2.IN_LOAD_UNLOAD_STATION_1 OR "DB4000_FIX_TABLE_POSITIONS".UNIT_02.FIXTURE_3.IN_LOAD_UNLOAD_STATION_1) AND NOT "DB7240_HARDWARE_SOFTWARE_ENABLE_DISABLE".DISABLE_FIXTURE.SW_UNIT_02_FIX_2_3_ENABLED) OR ("DB2031_CYCLES_GENERAL".CALIBRATION_CYCLE.CYCLE_SELECTED AND "DB2440_GLOBAL_DATA".GLOBAL_DATA.UNIT_02_ANY_FIX_CALIBRATION_MISS AND ("DB2440_GLOBAL_DATA".GLOBAL_DATA.FIX_IN_UNIT_02_STA_0_ANY_CALIBRATION_MISS OR ("DB8000_PART_STATUS".UNIT_02.STATION_1.PART_A.STATUS.MASTER_PART AND "DB8000_PART_STATUS".UNIT_02.STATION_1.PART_A.STATUS.PRESENT)))) AND "DB1251_PART_CYCLE_UNIT_02".U02_STA_1_COND_OK_STA_0_CYCLE AND "DB1251_PART_CYCLE_UNIT_02".U02_STA_2_COND_OK_STA_0_CYCLE AND "DB1251_PART_CYCLE_UNIT_02".U02_STA_3_COND_OK_STA_0_CYCLE AND "DB1251_PART_CYCLE_UNIT_02".U02_STA_4_COND_OK_STA_0_CYCLE AND NOT "DB7265_UNIT_02_ENABLE_DISABLE".DISABLED AND NOT "DB1281_UNIT_02_PART_CHECK_STATION_0".SEQUENCE.AUTO_REQUEST;
END_REGION

REGION Network 19: CYCLE UNIT 02 STATION 1
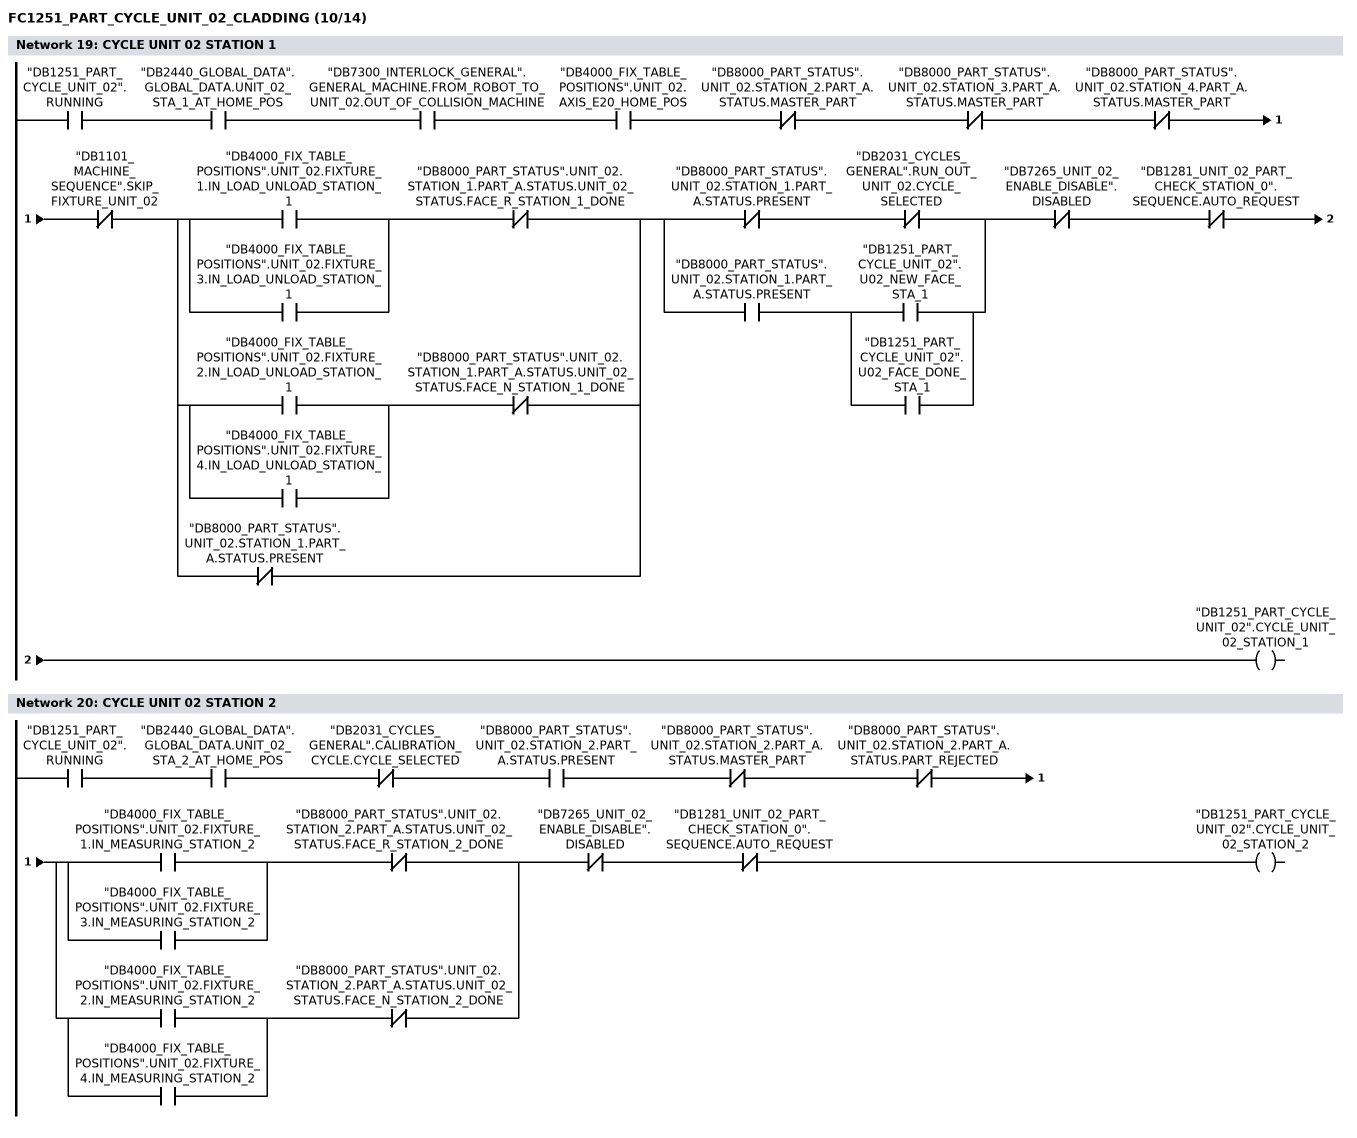
   RUNG wire#powerrail
      Contact( "DB1251_PART_CYCLE_UNIT_02".RUNNING )
      Contact( "DB2440_GLOBAL_DATA".GLOBAL_DATA.UNIT_02_STA_1_AT_HOME_POS )
      Contact( "DB7300_INTERLOCK_GENERAL".GENERAL_MACHINE.FROM_ROBOT_TO_UNIT_02.OUT_OF_COLLISION_MACHINE )
      Contact( "DB4000_FIX_TABLE_POSITIONS".UNIT_02.AXIS_E20_HOME_POS )
      I_Contact( "DB8000_PART_STATUS".UNIT_02.STATION_2.PART_A.STATUS.MASTER_PART )
      I_Contact( "DB8000_PART_STATUS".UNIT_02.STATION_3.PART_A.STATUS.MASTER_PART )
      I_Contact( "DB8000_PART_STATUS".UNIT_02.STATION_4.PART_A.STATUS.MASTER_PART )
      I_Contact( "DB1101_MACHINE_SEQUENCE".SKIP_FIXTURE_UNIT_02 )
      wire#w1
      Contact( "DB4000_FIX_TABLE_POSITIONS".UNIT_02.FIXTURE_1.IN_LOAD_UNLOAD_STATION_1 )
      wire#w2
      I_Contact( "DB8000_PART_STATUS".UNIT_02.STATION_1.PART_A.STATUS.UNIT_02_STATUS.FACE_R_STATION_1_DONE )
      wire#w3
      I_Contact( "DB8000_PART_STATUS".UNIT_02.STATION_1.PART_A.STATUS.PRESENT )
      I_Contact( "DB2031_CYCLES_GENERAL".RUN_OUT_UNIT_02.CYCLE_SELECTED )
      wire#w5
      I_Contact( "DB7265_UNIT_02_ENABLE_DISABLE".DISABLED )
      I_Contact( "DB1281_UNIT_02_PART_CHECK_STATION_0".SEQUENCE.AUTO_REQUEST )
      Coil( "DB1251_PART_CYCLE_UNIT_02".CYCLE_UNIT_02_STATION_1 )
   END_RUNG
   RUNG wire#w1
      Contact( "DB4000_FIX_TABLE_POSITIONS".UNIT_02.FIXTURE_3.IN_LOAD_UNLOAD_STATION_1 )
   END_RUNG wire#w2
   RUNG wire#w1
      Contact( "DB4000_FIX_TABLE_POSITIONS".UNIT_02.FIXTURE_2.IN_LOAD_UNLOAD_STATION_1 )
      wire#w4
      I_Contact( "DB8000_PART_STATUS".UNIT_02.STATION_1.PART_A.STATUS.UNIT_02_STATUS.FACE_N_STATION_1_DONE )
   END_RUNG wire#w3
   RUNG wire#w1
      Contact( "DB4000_FIX_TABLE_POSITIONS".UNIT_02.FIXTURE_4.IN_LOAD_UNLOAD_STATION_1 )
   END_RUNG wire#w4
   RUNG wire#w1
      I_Contact( "DB8000_PART_STATUS".UNIT_02.STATION_1.PART_A.STATUS.PRESENT )
   END_RUNG wire#w3
   RUNG wire#w3
      Contact( "DB8000_PART_STATUS".UNIT_02.STATION_1.PART_A.STATUS.PRESENT )
      wire#w6
      Contact( "DB1251_PART_CYCLE_UNIT_02".U02_NEW_FACE_STA_1 )
   END_RUNG wire#w5
   RUNG wire#w6
      Contact( "DB1251_PART_CYCLE_UNIT_02".U02_FACE_DONE_STA_1 )
   END_RUNG wire#w5
   // the same network as SCL:
   "DB1251_PART_CYCLE_UNIT_02".CYCLE_UNIT_02_STATION_1 := "DB1251_PART_CYCLE_UNIT_02".RUNNING AND "DB2440_GLOBAL_DATA".GLOBAL_DATA.UNIT_02_STA_1_AT_HOME_POS AND "DB7300_INTERLOCK_GENERAL".GENERAL_MACHINE.FROM_ROBOT_TO_UNIT_02.OUT_OF_COLLISION_MACHINE AND "DB4000_FIX_TABLE_POSITIONS".UNIT_02.AXIS_E20_HOME_POS AND NOT "DB8000_PART_STATUS".UNIT_02.STATION_2.PART_A.STATUS.MASTER_PART AND NOT "DB8000_PART_STATUS".UNIT_02.STATION_3.PART_A.STATUS.MASTER_PART AND NOT "DB8000_PART_STATUS".UNIT_02.STATION_4.PART_A.STATUS.MASTER_PART AND NOT "DB1101_MACHINE_SEQUENCE".SKIP_FIXTURE_UNIT_02 AND ((("DB4000_FIX_TABLE_POSITIONS".UNIT_02.FIXTURE_1.IN_LOAD_UNLOAD_STATION_1 OR "DB4000_FIX_TABLE_POSITIONS".UNIT_02.FIXTURE_3.IN_LOAD_UNLOAD_STATION_1) AND NOT "DB8000_PART_STATUS".UNIT_02.STATION_1.PART_A.STATUS.UNIT_02_STATUS.FACE_R_STATION_1_DONE) OR (("DB4000_FIX_TABLE_POSITIONS".UNIT_02.FIXTURE_2.IN_LOAD_UNLOAD_STATION_1 OR "DB4000_FIX_TABLE_POSITIONS".UNIT_02.FIXTURE_4.IN_LOAD_UNLOAD_STATION_1) AND NOT "DB8000_PART_STATUS".UNIT_02.STATION_1.PART_A.STATUS.UNIT_02_STATUS.FACE_N_STATION_1_DONE) OR NOT "DB8000_PART_STATUS".UNIT_02.STATION_1.PART_A.STATUS.PRESENT) AND ((NOT "DB8000_PART_STATUS".UNIT_02.STATION_1.PART_A.STATUS.PRESENT AND NOT "DB2031_CYCLES_GENERAL".RUN_OUT_UNIT_02.CYCLE_SELECTED) OR ("DB8000_PART_STATUS".UNIT_02.STATION_1.PART_A.STATUS.PRESENT AND ("DB1251_PART_CYCLE_UNIT_02".U02_NEW_FACE_STA_1 OR "DB1251_PART_CYCLE_UNIT_02".U02_FACE_DONE_STA_1))) AND NOT "DB7265_UNIT_02_ENABLE_DISABLE".DISABLED AND NOT "DB1281_UNIT_02_PART_CHECK_STATION_0".SEQUENCE.AUTO_REQUEST;
END_REGION

REGION Network 20: CYCLE UNIT 02 STATION 2
   RUNG wire#powerrail
      Contact( "DB1251_PART_CYCLE_UNIT_02".RUNNING )
      Contact( "DB2440_GLOBAL_DATA".GLOBAL_DATA.UNIT_02_STA_2_AT_HOME_POS )
      I_Contact( "DB2031_CYCLES_GENERAL".CALIBRATION_CYCLE.CYCLE_SELECTED )
      Contact( "DB8000_PART_STATUS".UNIT_02.STATION_2.PART_A.STATUS.PRESENT )
      I_Contact( "DB8000_PART_STATUS".UNIT_02.STATION_2.PART_A.STATUS.MASTER_PART )
      I_Contact( "DB8000_PART_STATUS".UNIT_02.STATION_2.PART_A.STATUS.PART_REJECTED )
      wire#w1
      Contact( "DB4000_FIX_TABLE_POSITIONS".UNIT_02.FIXTURE_1.IN_MEASURING_STATION_2 )
      wire#w2
      I_Contact( "DB8000_PART_STATUS".UNIT_02.STATION_2.PART_A.STATUS.UNIT_02_STATUS.FACE_R_STATION_2_DONE )
      wire#w3
      I_Contact( "DB7265_UNIT_02_ENABLE_DISABLE".DISABLED )
      I_Contact( "DB1281_UNIT_02_PART_CHECK_STATION_0".SEQUENCE.AUTO_REQUEST )
      Coil( "DB1251_PART_CYCLE_UNIT_02".CYCLE_UNIT_02_STATION_2 )
   END_RUNG
   RUNG wire#w1
      Contact( "DB4000_FIX_TABLE_POSITIONS".UNIT_02.FIXTURE_3.IN_MEASURING_STATION_2 )
   END_RUNG wire#w2
   RUNG wire#w1
      Contact( "DB4000_FIX_TABLE_POSITIONS".UNIT_02.FIXTURE_2.IN_MEASURING_STATION_2 )
      wire#w4
      I_Contact( "DB8000_PART_STATUS".UNIT_02.STATION_2.PART_A.STATUS.UNIT_02_STATUS.FACE_N_STATION_2_DONE )
   END_RUNG wire#w3
   RUNG wire#w1
      Contact( "DB4000_FIX_TABLE_POSITIONS".UNIT_02.FIXTURE_4.IN_MEASURING_STATION_2 )
   END_RUNG wire#w4
   // the same network as SCL:
   "DB1251_PART_CYCLE_UNIT_02".CYCLE_UNIT_02_STATION_2 := "DB1251_PART_CYCLE_UNIT_02".RUNNING AND "DB2440_GLOBAL_DATA".GLOBAL_DATA.UNIT_02_STA_2_AT_HOME_POS AND NOT "DB2031_CYCLES_GENERAL".CALIBRATION_CYCLE.CYCLE_SELECTED AND "DB8000_PART_STATUS".UNIT_02.STATION_2.PART_A.STATUS.PRESENT AND NOT "DB8000_PART_STATUS".UNIT_02.STATION_2.PART_A.STATUS.MASTER_PART AND NOT "DB8000_PART_STATUS".UNIT_02.STATION_2.PART_A.STATUS.PART_REJECTED AND ((("DB4000_FIX_TABLE_POSITIONS".UNIT_02.FIXTURE_1.IN_MEASURING_STATION_2 OR "DB4000_FIX_TABLE_POSITIONS".UNIT_02.FIXTURE_3.IN_MEASURING_STATION_2) AND NOT "DB8000_PART_STATUS".UNIT_02.STATION_2.PART_A.STATUS.UNIT_02_STATUS.FACE_R_STATION_2_DONE) OR (("DB4000_FIX_TABLE_POSITIONS".UNIT_02.FIXTURE_2.IN_MEASURING_STATION_2 OR "DB4000_FIX_TABLE_POSITIONS".UNIT_02.FIXTURE_4.IN_MEASURING_STATION_2) AND NOT "DB8000_PART_STATUS".UNIT_02.STATION_2.PART_A.STATUS.UNIT_02_STATUS.FACE_N_STATION_2_DONE)) AND NOT "DB7265_UNIT_02_ENABLE_DISABLE".DISABLED AND NOT "DB1281_UNIT_02_PART_CHECK_STATION_0".SEQUENCE.AUTO_REQUEST;
END_REGION

REGION Network 21: CYCLE UNIT 02 STATION 3
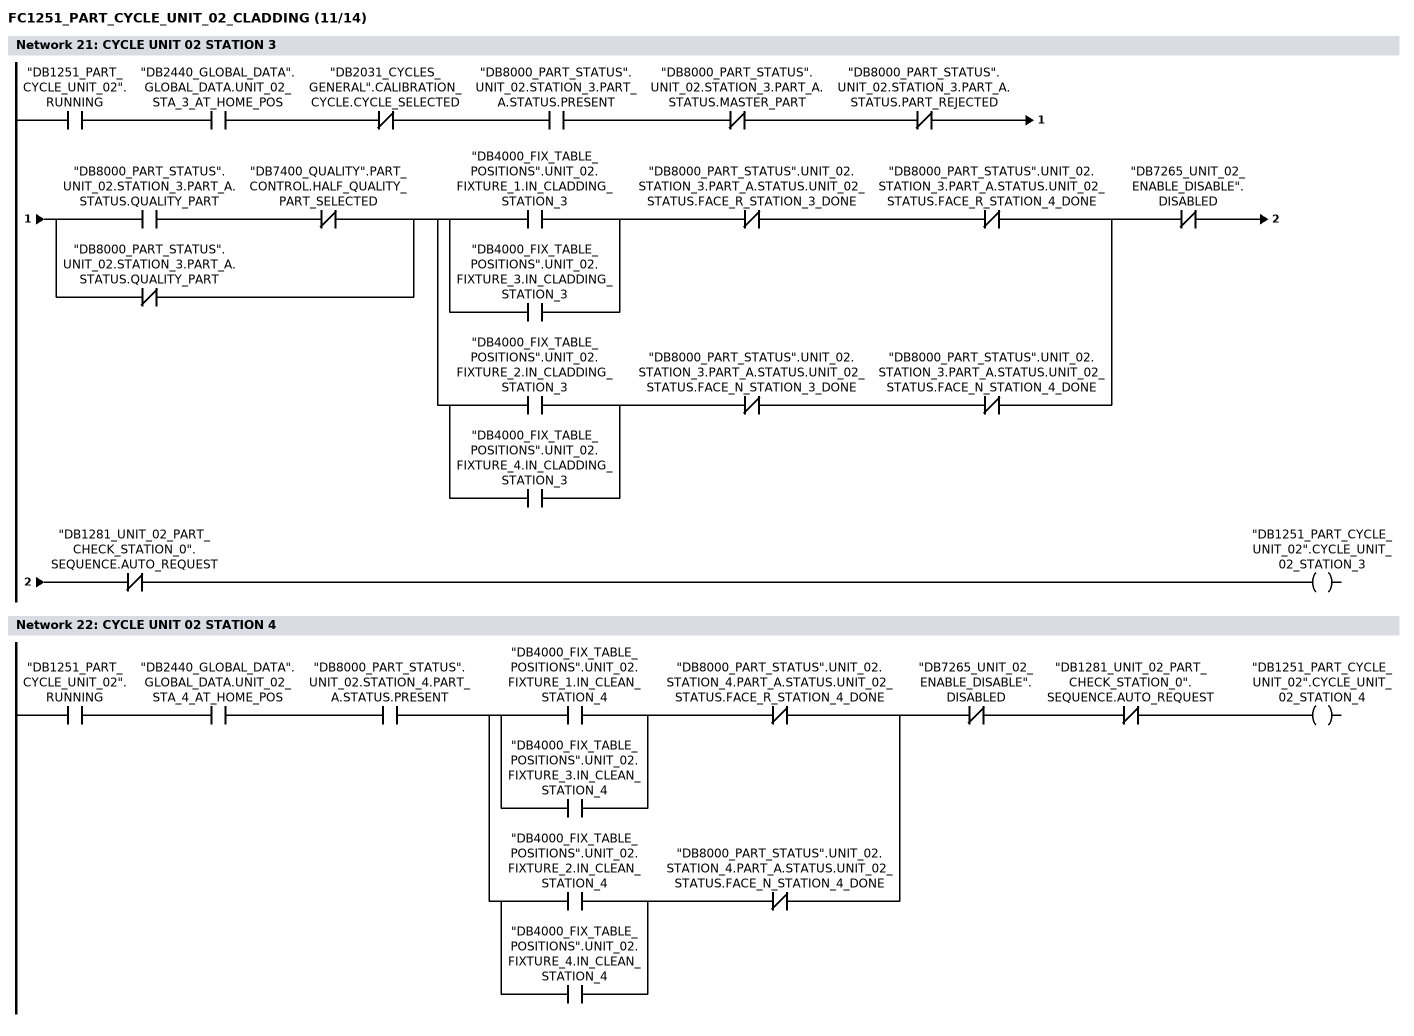
   RUNG wire#powerrail
      Contact( "DB1251_PART_CYCLE_UNIT_02".RUNNING )
      Contact( "DB2440_GLOBAL_DATA".GLOBAL_DATA.UNIT_02_STA_3_AT_HOME_POS )
      I_Contact( "DB2031_CYCLES_GENERAL".CALIBRATION_CYCLE.CYCLE_SELECTED )
      Contact( "DB8000_PART_STATUS".UNIT_02.STATION_3.PART_A.STATUS.PRESENT )
      I_Contact( "DB8000_PART_STATUS".UNIT_02.STATION_3.PART_A.STATUS.MASTER_PART )
      I_Contact( "DB8000_PART_STATUS".UNIT_02.STATION_3.PART_A.STATUS.PART_REJECTED )
      wire#w1
      Contact( "DB8000_PART_STATUS".UNIT_02.STATION_3.PART_A.STATUS.QUALITY_PART )
      I_Contact( "DB7400_QUALITY".PART_CONTROL.HALF_QUALITY_PART_SELECTED )
      wire#w2
      Contact( "DB4000_FIX_TABLE_POSITIONS".UNIT_02.FIXTURE_1.IN_CLADDING_STATION_3 )
      wire#w3
      I_Contact( "DB8000_PART_STATUS".UNIT_02.STATION_3.PART_A.STATUS.UNIT_02_STATUS.FACE_R_STATION_3_DONE )
      I_Contact( "DB8000_PART_STATUS".UNIT_02.STATION_3.PART_A.STATUS.UNIT_02_STATUS.FACE_R_STATION_4_DONE )
      wire#w4
      I_Contact( "DB7265_UNIT_02_ENABLE_DISABLE".DISABLED )
      I_Contact( "DB1281_UNIT_02_PART_CHECK_STATION_0".SEQUENCE.AUTO_REQUEST )
      Coil( "DB1251_PART_CYCLE_UNIT_02".CYCLE_UNIT_02_STATION_3 )
   END_RUNG
   RUNG wire#w1
      I_Contact( "DB8000_PART_STATUS".UNIT_02.STATION_3.PART_A.STATUS.QUALITY_PART )
   END_RUNG wire#w2
   RUNG wire#w2
      Contact( "DB4000_FIX_TABLE_POSITIONS".UNIT_02.FIXTURE_3.IN_CLADDING_STATION_3 )
   END_RUNG wire#w3
   RUNG wire#w2
      Contact( "DB4000_FIX_TABLE_POSITIONS".UNIT_02.FIXTURE_2.IN_CLADDING_STATION_3 )
      wire#w5
      I_Contact( "DB8000_PART_STATUS".UNIT_02.STATION_3.PART_A.STATUS.UNIT_02_STATUS.FACE_N_STATION_3_DONE )
      I_Contact( "DB8000_PART_STATUS".UNIT_02.STATION_3.PART_A.STATUS.UNIT_02_STATUS.FACE_N_STATION_4_DONE )
   END_RUNG wire#w4
   RUNG wire#w2
      Contact( "DB4000_FIX_TABLE_POSITIONS".UNIT_02.FIXTURE_4.IN_CLADDING_STATION_3 )
   END_RUNG wire#w5
   // the same network as SCL:
   "DB1251_PART_CYCLE_UNIT_02".CYCLE_UNIT_02_STATION_3 := "DB1251_PART_CYCLE_UNIT_02".RUNNING AND "DB2440_GLOBAL_DATA".GLOBAL_DATA.UNIT_02_STA_3_AT_HOME_POS AND NOT "DB2031_CYCLES_GENERAL".CALIBRATION_CYCLE.CYCLE_SELECTED AND "DB8000_PART_STATUS".UNIT_02.STATION_3.PART_A.STATUS.PRESENT AND NOT "DB8000_PART_STATUS".UNIT_02.STATION_3.PART_A.STATUS.MASTER_PART AND NOT "DB8000_PART_STATUS".UNIT_02.STATION_3.PART_A.STATUS.PART_REJECTED AND (("DB8000_PART_STATUS".UNIT_02.STATION_3.PART_A.STATUS.QUALITY_PART AND NOT "DB7400_QUALITY".PART_CONTROL.HALF_QUALITY_PART_SELECTED) OR NOT "DB8000_PART_STATUS".UNIT_02.STATION_3.PART_A.STATUS.QUALITY_PART) AND ((("DB4000_FIX_TABLE_POSITIONS".UNIT_02.FIXTURE_1.IN_CLADDING_STATION_3 OR "DB4000_FIX_TABLE_POSITIONS".UNIT_02.FIXTURE_3.IN_CLADDING_STATION_3) AND NOT "DB8000_PART_STATUS".UNIT_02.STATION_3.PART_A.STATUS.UNIT_02_STATUS.FACE_R_STATION_3_DONE AND NOT "DB8000_PART_STATUS".UNIT_02.STATION_3.PART_A.STATUS.UNIT_02_STATUS.FACE_R_STATION_4_DONE) OR (("DB4000_FIX_TABLE_POSITIONS".UNIT_02.FIXTURE_2.IN_CLADDING_STATION_3 OR "DB4000_FIX_TABLE_POSITIONS".UNIT_02.FIXTURE_4.IN_CLADDING_STATION_3) AND NOT "DB8000_PART_STATUS".UNIT_02.STATION_3.PART_A.STATUS.UNIT_02_STATUS.FACE_N_STATION_3_DONE AND NOT "DB8000_PART_STATUS".UNIT_02.STATION_3.PART_A.STATUS.UNIT_02_STATUS.FACE_N_STATION_4_DONE)) AND NOT "DB7265_UNIT_02_ENABLE_DISABLE".DISABLED AND NOT "DB1281_UNIT_02_PART_CHECK_STATION_0".SEQUENCE.AUTO_REQUEST;
END_REGION

REGION Network 22: CYCLE UNIT 02 STATION 4
   RUNG wire#powerrail
      Contact( "DB1251_PART_CYCLE_UNIT_02".RUNNING )
      Contact( "DB2440_GLOBAL_DATA".GLOBAL_DATA.UNIT_02_STA_4_AT_HOME_POS )
      Contact( "DB8000_PART_STATUS".UNIT_02.STATION_4.PART_A.STATUS.PRESENT )
      wire#w1
      Contact( "DB4000_FIX_TABLE_POSITIONS".UNIT_02.FIXTURE_1.IN_CLEAN_STATION_4 )
      wire#w2
      I_Contact( "DB8000_PART_STATUS".UNIT_02.STATION_4.PART_A.STATUS.UNIT_02_STATUS.FACE_R_STATION_4_DONE )
      wire#w3
      I_Contact( "DB7265_UNIT_02_ENABLE_DISABLE".DISABLED )
      I_Contact( "DB1281_UNIT_02_PART_CHECK_STATION_0".SEQUENCE.AUTO_REQUEST )
      Coil( "DB1251_PART_CYCLE_UNIT_02".CYCLE_UNIT_02_STATION_4 )
   END_RUNG
   RUNG wire#w1
      Contact( "DB4000_FIX_TABLE_POSITIONS".UNIT_02.FIXTURE_3.IN_CLEAN_STATION_4 )
   END_RUNG wire#w2
   RUNG wire#w1
      Contact( "DB4000_FIX_TABLE_POSITIONS".UNIT_02.FIXTURE_2.IN_CLEAN_STATION_4 )
      wire#w4
      I_Contact( "DB8000_PART_STATUS".UNIT_02.STATION_4.PART_A.STATUS.UNIT_02_STATUS.FACE_N_STATION_4_DONE )
   END_RUNG wire#w3
   RUNG wire#w1
      Contact( "DB4000_FIX_TABLE_POSITIONS".UNIT_02.FIXTURE_4.IN_CLEAN_STATION_4 )
   END_RUNG wire#w4
   // the same network as SCL:
   "DB1251_PART_CYCLE_UNIT_02".CYCLE_UNIT_02_STATION_4 := "DB1251_PART_CYCLE_UNIT_02".RUNNING AND "DB2440_GLOBAL_DATA".GLOBAL_DATA.UNIT_02_STA_4_AT_HOME_POS AND "DB8000_PART_STATUS".UNIT_02.STATION_4.PART_A.STATUS.PRESENT AND ((("DB4000_FIX_TABLE_POSITIONS".UNIT_02.FIXTURE_1.IN_CLEAN_STATION_4 OR "DB4000_FIX_TABLE_POSITIONS".UNIT_02.FIXTURE_3.IN_CLEAN_STATION_4) AND NOT "DB8000_PART_STATUS".UNIT_02.STATION_4.PART_A.STATUS.UNIT_02_STATUS.FACE_R_STATION_4_DONE) OR (("DB4000_FIX_TABLE_POSITIONS".UNIT_02.FIXTURE_2.IN_CLEAN_STATION_4 OR "DB4000_FIX_TABLE_POSITIONS".UNIT_02.FIXTURE_4.IN_CLEAN_STATION_4) AND NOT "DB8000_PART_STATUS".UNIT_02.STATION_4.PART_A.STATUS.UNIT_02_STATUS.FACE_N_STATION_4_DONE)) AND NOT "DB7265_UNIT_02_ENABLE_DISABLE".DISABLED AND NOT "DB1281_UNIT_02_PART_CHECK_STATION_0".SEQUENCE.AUTO_REQUEST;
END_REGION

REGION Network 23: UNIT 02 STATION 2 CALIBRATION
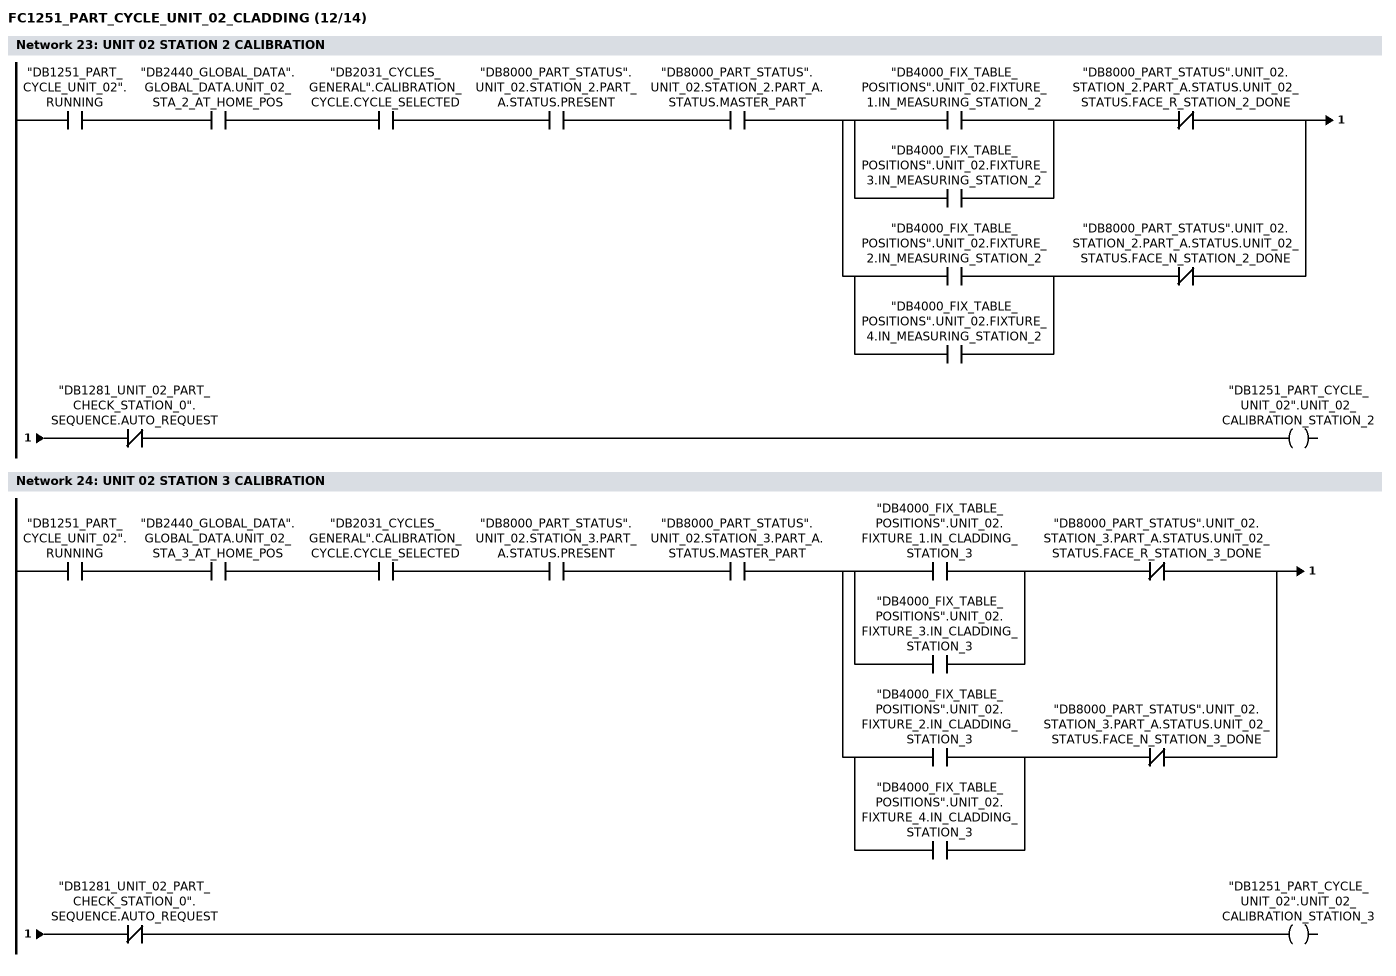
   RUNG wire#powerrail
      Contact( "DB1251_PART_CYCLE_UNIT_02".RUNNING )
      Contact( "DB2440_GLOBAL_DATA".GLOBAL_DATA.UNIT_02_STA_2_AT_HOME_POS )
      Contact( "DB2031_CYCLES_GENERAL".CALIBRATION_CYCLE.CYCLE_SELECTED )
      Contact( "DB8000_PART_STATUS".UNIT_02.STATION_2.PART_A.STATUS.PRESENT )
      Contact( "DB8000_PART_STATUS".UNIT_02.STATION_2.PART_A.STATUS.MASTER_PART )
      wire#w1
      Contact( "DB4000_FIX_TABLE_POSITIONS".UNIT_02.FIXTURE_1.IN_MEASURING_STATION_2 )
      wire#w2
      I_Contact( "DB8000_PART_STATUS".UNIT_02.STATION_2.PART_A.STATUS.UNIT_02_STATUS.FACE_R_STATION_2_DONE )
      wire#w3
      I_Contact( "DB1281_UNIT_02_PART_CHECK_STATION_0".SEQUENCE.AUTO_REQUEST )
      Coil( "DB1251_PART_CYCLE_UNIT_02".UNIT_02_CALIBRATION_STATION_2 )
   END_RUNG
   RUNG wire#w1
      Contact( "DB4000_FIX_TABLE_POSITIONS".UNIT_02.FIXTURE_3.IN_MEASURING_STATION_2 )
   END_RUNG wire#w2
   RUNG wire#w1
      Contact( "DB4000_FIX_TABLE_POSITIONS".UNIT_02.FIXTURE_2.IN_MEASURING_STATION_2 )
      wire#w4
      I_Contact( "DB8000_PART_STATUS".UNIT_02.STATION_2.PART_A.STATUS.UNIT_02_STATUS.FACE_N_STATION_2_DONE )
   END_RUNG wire#w3
   RUNG wire#w1
      Contact( "DB4000_FIX_TABLE_POSITIONS".UNIT_02.FIXTURE_4.IN_MEASURING_STATION_2 )
   END_RUNG wire#w4
   // the same network as SCL:
   "DB1251_PART_CYCLE_UNIT_02".UNIT_02_CALIBRATION_STATION_2 := "DB1251_PART_CYCLE_UNIT_02".RUNNING AND "DB2440_GLOBAL_DATA".GLOBAL_DATA.UNIT_02_STA_2_AT_HOME_POS AND "DB2031_CYCLES_GENERAL".CALIBRATION_CYCLE.CYCLE_SELECTED AND "DB8000_PART_STATUS".UNIT_02.STATION_2.PART_A.STATUS.PRESENT AND "DB8000_PART_STATUS".UNIT_02.STATION_2.PART_A.STATUS.MASTER_PART AND ((("DB4000_FIX_TABLE_POSITIONS".UNIT_02.FIXTURE_1.IN_MEASURING_STATION_2 OR "DB4000_FIX_TABLE_POSITIONS".UNIT_02.FIXTURE_3.IN_MEASURING_STATION_2) AND NOT "DB8000_PART_STATUS".UNIT_02.STATION_2.PART_A.STATUS.UNIT_02_STATUS.FACE_R_STATION_2_DONE) OR (("DB4000_FIX_TABLE_POSITIONS".UNIT_02.FIXTURE_2.IN_MEASURING_STATION_2 OR "DB4000_FIX_TABLE_POSITIONS".UNIT_02.FIXTURE_4.IN_MEASURING_STATION_2) AND NOT "DB8000_PART_STATUS".UNIT_02.STATION_2.PART_A.STATUS.UNIT_02_STATUS.FACE_N_STATION_2_DONE)) AND NOT "DB1281_UNIT_02_PART_CHECK_STATION_0".SEQUENCE.AUTO_REQUEST;
END_REGION

REGION Network 24: UNIT 02 STATION 3 CALIBRATION
   RUNG wire#powerrail
      Contact( "DB1251_PART_CYCLE_UNIT_02".RUNNING )
      Contact( "DB2440_GLOBAL_DATA".GLOBAL_DATA.UNIT_02_STA_3_AT_HOME_POS )
      Contact( "DB2031_CYCLES_GENERAL".CALIBRATION_CYCLE.CYCLE_SELECTED )
      Contact( "DB8000_PART_STATUS".UNIT_02.STATION_3.PART_A.STATUS.PRESENT )
      Contact( "DB8000_PART_STATUS".UNIT_02.STATION_3.PART_A.STATUS.MASTER_PART )
      wire#w1
      Contact( "DB4000_FIX_TABLE_POSITIONS".UNIT_02.FIXTURE_1.IN_CLADDING_STATION_3 )
      wire#w2
      I_Contact( "DB8000_PART_STATUS".UNIT_02.STATION_3.PART_A.STATUS.UNIT_02_STATUS.FACE_R_STATION_3_DONE )
      wire#w3
      I_Contact( "DB1281_UNIT_02_PART_CHECK_STATION_0".SEQUENCE.AUTO_REQUEST )
      Coil( "DB1251_PART_CYCLE_UNIT_02".UNIT_02_CALIBRATION_STATION_3 )
   END_RUNG
   RUNG wire#w1
      Contact( "DB4000_FIX_TABLE_POSITIONS".UNIT_02.FIXTURE_3.IN_CLADDING_STATION_3 )
   END_RUNG wire#w2
   RUNG wire#w1
      Contact( "DB4000_FIX_TABLE_POSITIONS".UNIT_02.FIXTURE_2.IN_CLADDING_STATION_3 )
      wire#w4
      I_Contact( "DB8000_PART_STATUS".UNIT_02.STATION_3.PART_A.STATUS.UNIT_02_STATUS.FACE_N_STATION_3_DONE )
   END_RUNG wire#w3
   RUNG wire#w1
      Contact( "DB4000_FIX_TABLE_POSITIONS".UNIT_02.FIXTURE_4.IN_CLADDING_STATION_3 )
   END_RUNG wire#w4
   // the same network as SCL:
   "DB1251_PART_CYCLE_UNIT_02".UNIT_02_CALIBRATION_STATION_3 := "DB1251_PART_CYCLE_UNIT_02".RUNNING AND "DB2440_GLOBAL_DATA".GLOBAL_DATA.UNIT_02_STA_3_AT_HOME_POS AND "DB2031_CYCLES_GENERAL".CALIBRATION_CYCLE.CYCLE_SELECTED AND "DB8000_PART_STATUS".UNIT_02.STATION_3.PART_A.STATUS.PRESENT AND "DB8000_PART_STATUS".UNIT_02.STATION_3.PART_A.STATUS.MASTER_PART AND ((("DB4000_FIX_TABLE_POSITIONS".UNIT_02.FIXTURE_1.IN_CLADDING_STATION_3 OR "DB4000_FIX_TABLE_POSITIONS".UNIT_02.FIXTURE_3.IN_CLADDING_STATION_3) AND NOT "DB8000_PART_STATUS".UNIT_02.STATION_3.PART_A.STATUS.UNIT_02_STATUS.FACE_R_STATION_3_DONE) OR (("DB4000_FIX_TABLE_POSITIONS".UNIT_02.FIXTURE_2.IN_CLADDING_STATION_3 OR "DB4000_FIX_TABLE_POSITIONS".UNIT_02.FIXTURE_4.IN_CLADDING_STATION_3) AND NOT "DB8000_PART_STATUS".UNIT_02.STATION_3.PART_A.STATUS.UNIT_02_STATUS.FACE_N_STATION_3_DONE)) AND NOT "DB1281_UNIT_02_PART_CHECK_STATION_0".SEQUENCE.AUTO_REQUEST;
END_REGION

REGION Network 25: CYCLE UNIT 02 STATION 2 MASTER MEASUREMENT
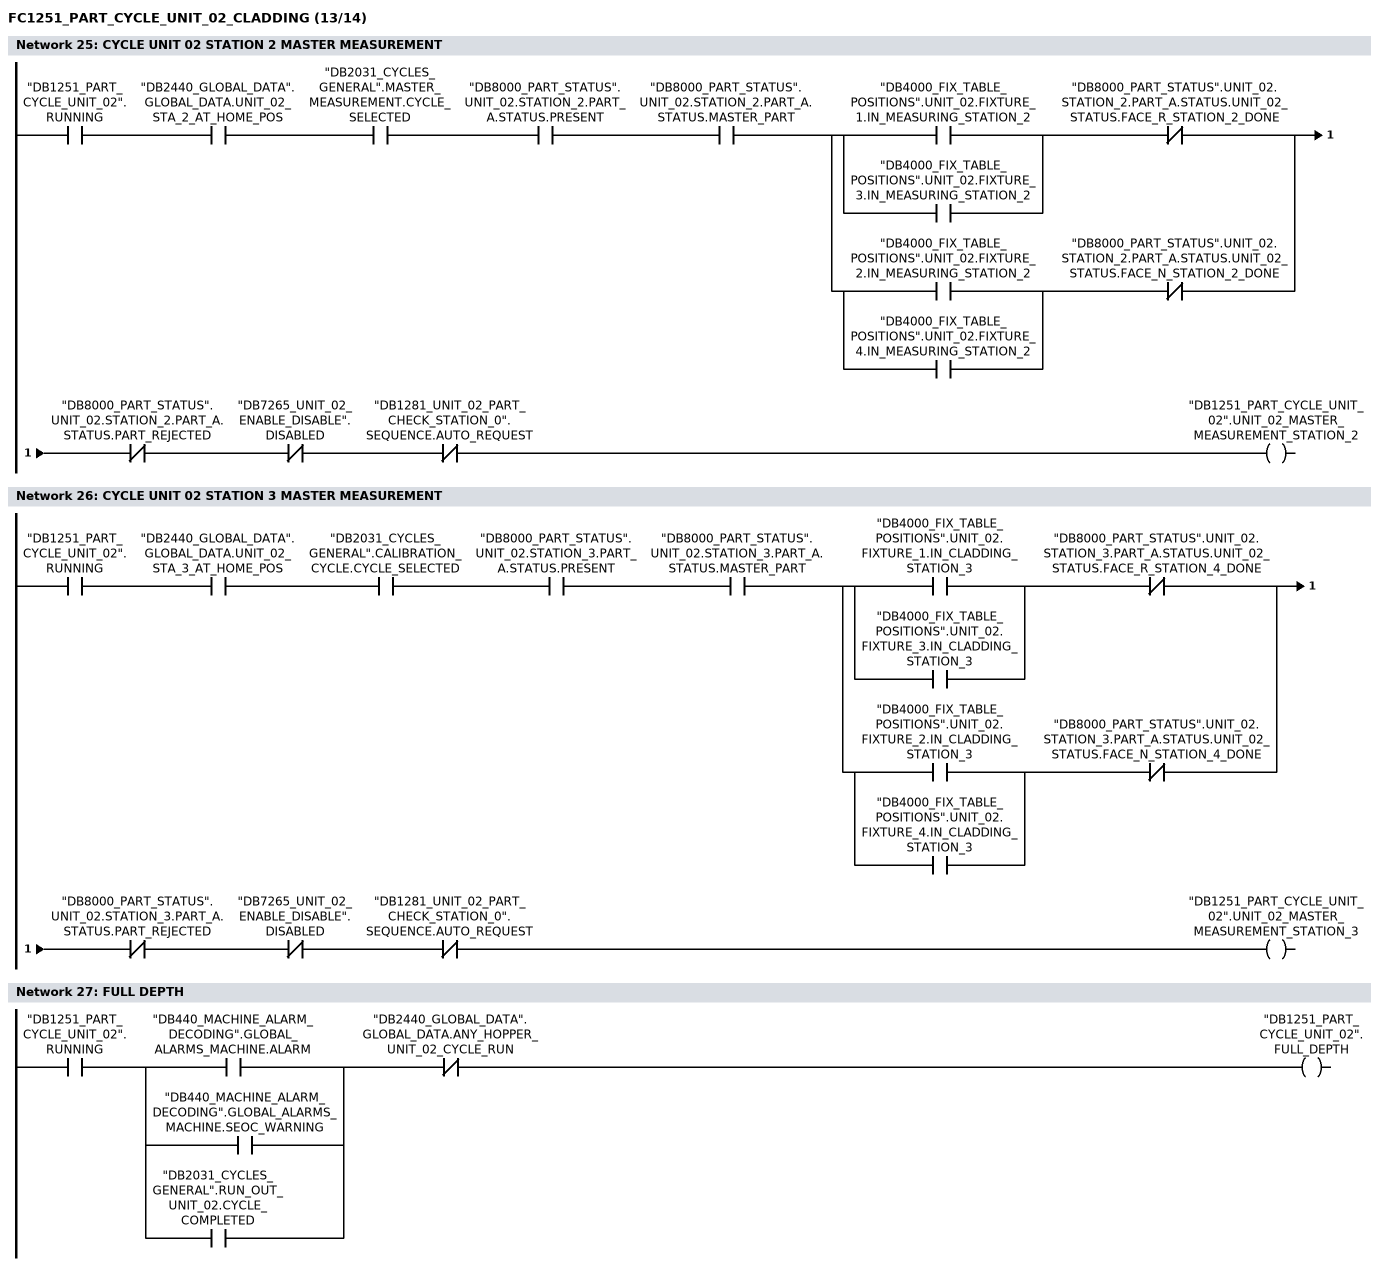
   RUNG wire#powerrail
      Contact( "DB1251_PART_CYCLE_UNIT_02".RUNNING )
      Contact( "DB2440_GLOBAL_DATA".GLOBAL_DATA.UNIT_02_STA_2_AT_HOME_POS )
      Contact( "DB2031_CYCLES_GENERAL".MASTER_MEASUREMENT.CYCLE_SELECTED )
      Contact( "DB8000_PART_STATUS".UNIT_02.STATION_2.PART_A.STATUS.PRESENT )
      Contact( "DB8000_PART_STATUS".UNIT_02.STATION_2.PART_A.STATUS.MASTER_PART )
      wire#w1
      Contact( "DB4000_FIX_TABLE_POSITIONS".UNIT_02.FIXTURE_1.IN_MEASURING_STATION_2 )
      wire#w2
      I_Contact( "DB8000_PART_STATUS".UNIT_02.STATION_2.PART_A.STATUS.UNIT_02_STATUS.FACE_R_STATION_2_DONE )
      wire#w3
      I_Contact( "DB8000_PART_STATUS".UNIT_02.STATION_2.PART_A.STATUS.PART_REJECTED )
      I_Contact( "DB7265_UNIT_02_ENABLE_DISABLE".DISABLED )
      I_Contact( "DB1281_UNIT_02_PART_CHECK_STATION_0".SEQUENCE.AUTO_REQUEST )
      Coil( "DB1251_PART_CYCLE_UNIT_02".UNIT_02_MASTER_MEASUREMENT_STATION_2 )
   END_RUNG
   RUNG wire#w1
      Contact( "DB4000_FIX_TABLE_POSITIONS".UNIT_02.FIXTURE_3.IN_MEASURING_STATION_2 )
   END_RUNG wire#w2
   RUNG wire#w1
      Contact( "DB4000_FIX_TABLE_POSITIONS".UNIT_02.FIXTURE_2.IN_MEASURING_STATION_2 )
      wire#w4
      I_Contact( "DB8000_PART_STATUS".UNIT_02.STATION_2.PART_A.STATUS.UNIT_02_STATUS.FACE_N_STATION_2_DONE )
   END_RUNG wire#w3
   RUNG wire#w1
      Contact( "DB4000_FIX_TABLE_POSITIONS".UNIT_02.FIXTURE_4.IN_MEASURING_STATION_2 )
   END_RUNG wire#w4
   // the same network as SCL:
   "DB1251_PART_CYCLE_UNIT_02".UNIT_02_MASTER_MEASUREMENT_STATION_2 := "DB1251_PART_CYCLE_UNIT_02".RUNNING AND "DB2440_GLOBAL_DATA".GLOBAL_DATA.UNIT_02_STA_2_AT_HOME_POS AND "DB2031_CYCLES_GENERAL".MASTER_MEASUREMENT.CYCLE_SELECTED AND "DB8000_PART_STATUS".UNIT_02.STATION_2.PART_A.STATUS.PRESENT AND "DB8000_PART_STATUS".UNIT_02.STATION_2.PART_A.STATUS.MASTER_PART AND ((("DB4000_FIX_TABLE_POSITIONS".UNIT_02.FIXTURE_1.IN_MEASURING_STATION_2 OR "DB4000_FIX_TABLE_POSITIONS".UNIT_02.FIXTURE_3.IN_MEASURING_STATION_2) AND NOT "DB8000_PART_STATUS".UNIT_02.STATION_2.PART_A.STATUS.UNIT_02_STATUS.FACE_R_STATION_2_DONE) OR (("DB4000_FIX_TABLE_POSITIONS".UNIT_02.FIXTURE_2.IN_MEASURING_STATION_2 OR "DB4000_FIX_TABLE_POSITIONS".UNIT_02.FIXTURE_4.IN_MEASURING_STATION_2) AND NOT "DB8000_PART_STATUS".UNIT_02.STATION_2.PART_A.STATUS.UNIT_02_STATUS.FACE_N_STATION_2_DONE)) AND NOT "DB8000_PART_STATUS".UNIT_02.STATION_2.PART_A.STATUS.PART_REJECTED AND NOT "DB7265_UNIT_02_ENABLE_DISABLE".DISABLED AND NOT "DB1281_UNIT_02_PART_CHECK_STATION_0".SEQUENCE.AUTO_REQUEST;
END_REGION

REGION Network 26: CYCLE UNIT 02 STATION 3 MASTER MEASUREMENT
   RUNG wire#powerrail
      Contact( "DB1251_PART_CYCLE_UNIT_02".RUNNING )
      Contact( "DB2440_GLOBAL_DATA".GLOBAL_DATA.UNIT_02_STA_3_AT_HOME_POS )
      Contact( "DB2031_CYCLES_GENERAL".CALIBRATION_CYCLE.CYCLE_SELECTED )
      Contact( "DB8000_PART_STATUS".UNIT_02.STATION_3.PART_A.STATUS.PRESENT )
      Contact( "DB8000_PART_STATUS".UNIT_02.STATION_3.PART_A.STATUS.MASTER_PART )
      wire#w1
      Contact( "DB4000_FIX_TABLE_POSITIONS".UNIT_02.FIXTURE_1.IN_CLADDING_STATION_3 )
      wire#w2
      I_Contact( "DB8000_PART_STATUS".UNIT_02.STATION_3.PART_A.STATUS.UNIT_02_STATUS.FACE_R_STATION_4_DONE )
      wire#w3
      I_Contact( "DB8000_PART_STATUS".UNIT_02.STATION_3.PART_A.STATUS.PART_REJECTED )
      I_Contact( "DB7265_UNIT_02_ENABLE_DISABLE".DISABLED )
      I_Contact( "DB1281_UNIT_02_PART_CHECK_STATION_0".SEQUENCE.AUTO_REQUEST )
      Coil( "DB1251_PART_CYCLE_UNIT_02".UNIT_02_MASTER_MEASUREMENT_STATION_3 )
   END_RUNG
   RUNG wire#w1
      Contact( "DB4000_FIX_TABLE_POSITIONS".UNIT_02.FIXTURE_3.IN_CLADDING_STATION_3 )
   END_RUNG wire#w2
   RUNG wire#w1
      Contact( "DB4000_FIX_TABLE_POSITIONS".UNIT_02.FIXTURE_2.IN_CLADDING_STATION_3 )
      wire#w4
      I_Contact( "DB8000_PART_STATUS".UNIT_02.STATION_3.PART_A.STATUS.UNIT_02_STATUS.FACE_N_STATION_4_DONE )
   END_RUNG wire#w3
   RUNG wire#w1
      Contact( "DB4000_FIX_TABLE_POSITIONS".UNIT_02.FIXTURE_4.IN_CLADDING_STATION_3 )
   END_RUNG wire#w4
   // the same network as SCL:
   "DB1251_PART_CYCLE_UNIT_02".UNIT_02_MASTER_MEASUREMENT_STATION_3 := "DB1251_PART_CYCLE_UNIT_02".RUNNING AND "DB2440_GLOBAL_DATA".GLOBAL_DATA.UNIT_02_STA_3_AT_HOME_POS AND "DB2031_CYCLES_GENERAL".CALIBRATION_CYCLE.CYCLE_SELECTED AND "DB8000_PART_STATUS".UNIT_02.STATION_3.PART_A.STATUS.PRESENT AND "DB8000_PART_STATUS".UNIT_02.STATION_3.PART_A.STATUS.MASTER_PART AND ((("DB4000_FIX_TABLE_POSITIONS".UNIT_02.FIXTURE_1.IN_CLADDING_STATION_3 OR "DB4000_FIX_TABLE_POSITIONS".UNIT_02.FIXTURE_3.IN_CLADDING_STATION_3) AND NOT "DB8000_PART_STATUS".UNIT_02.STATION_3.PART_A.STATUS.UNIT_02_STATUS.FACE_R_STATION_4_DONE) OR (("DB4000_FIX_TABLE_POSITIONS".UNIT_02.FIXTURE_2.IN_CLADDING_STATION_3 OR "DB4000_FIX_TABLE_POSITIONS".UNIT_02.FIXTURE_4.IN_CLADDING_STATION_3) AND NOT "DB8000_PART_STATUS".UNIT_02.STATION_3.PART_A.STATUS.UNIT_02_STATUS.FACE_N_STATION_4_DONE)) AND NOT "DB8000_PART_STATUS".UNIT_02.STATION_3.PART_A.STATUS.PART_REJECTED AND NOT "DB7265_UNIT_02_ENABLE_DISABLE".DISABLED AND NOT "DB1281_UNIT_02_PART_CHECK_STATION_0".SEQUENCE.AUTO_REQUEST;
END_REGION

REGION Network 27: FULL DEPTH
   RUNG wire#powerrail
      Contact( "DB1251_PART_CYCLE_UNIT_02".RUNNING )
      wire#w1
      Contact( "DB440_MACHINE_ALARM_DECODING".GLOBAL_ALARMS_MACHINE.ALARM )
      wire#w2
      I_Contact( "DB2440_GLOBAL_DATA".GLOBAL_DATA.ANY_HOPPER_UNIT_02_CYCLE_RUN )
      Coil( "DB1251_PART_CYCLE_UNIT_02".FULL_DEPTH )
   END_RUNG
   RUNG wire#w1
      Contact( "DB440_MACHINE_ALARM_DECODING".GLOBAL_ALARMS_MACHINE.SEOC_WARNING )
   END_RUNG wire#w2
   RUNG wire#w1
      Contact( "DB2031_CYCLES_GENERAL".RUN_OUT_UNIT_02.CYCLE_COMPLETED )
   END_RUNG wire#w2
   // the same network as SCL:
   "DB1251_PART_CYCLE_UNIT_02".FULL_DEPTH := "DB1251_PART_CYCLE_UNIT_02".RUNNING AND ("DB440_MACHINE_ALARM_DECODING".GLOBAL_ALARMS_MACHINE.ALARM OR "DB440_MACHINE_ALARM_DECODING".GLOBAL_ALARMS_MACHINE.SEOC_WARNING OR "DB2031_CYCLES_GENERAL".RUN_OUT_UNIT_02.CYCLE_COMPLETED) AND NOT "DB2440_GLOBAL_DATA".GLOBAL_DATA.ANY_HOPPER_UNIT_02_CYCLE_RUN;
END_REGION

REGION Network 28: TIME EXCEEDED ALARM
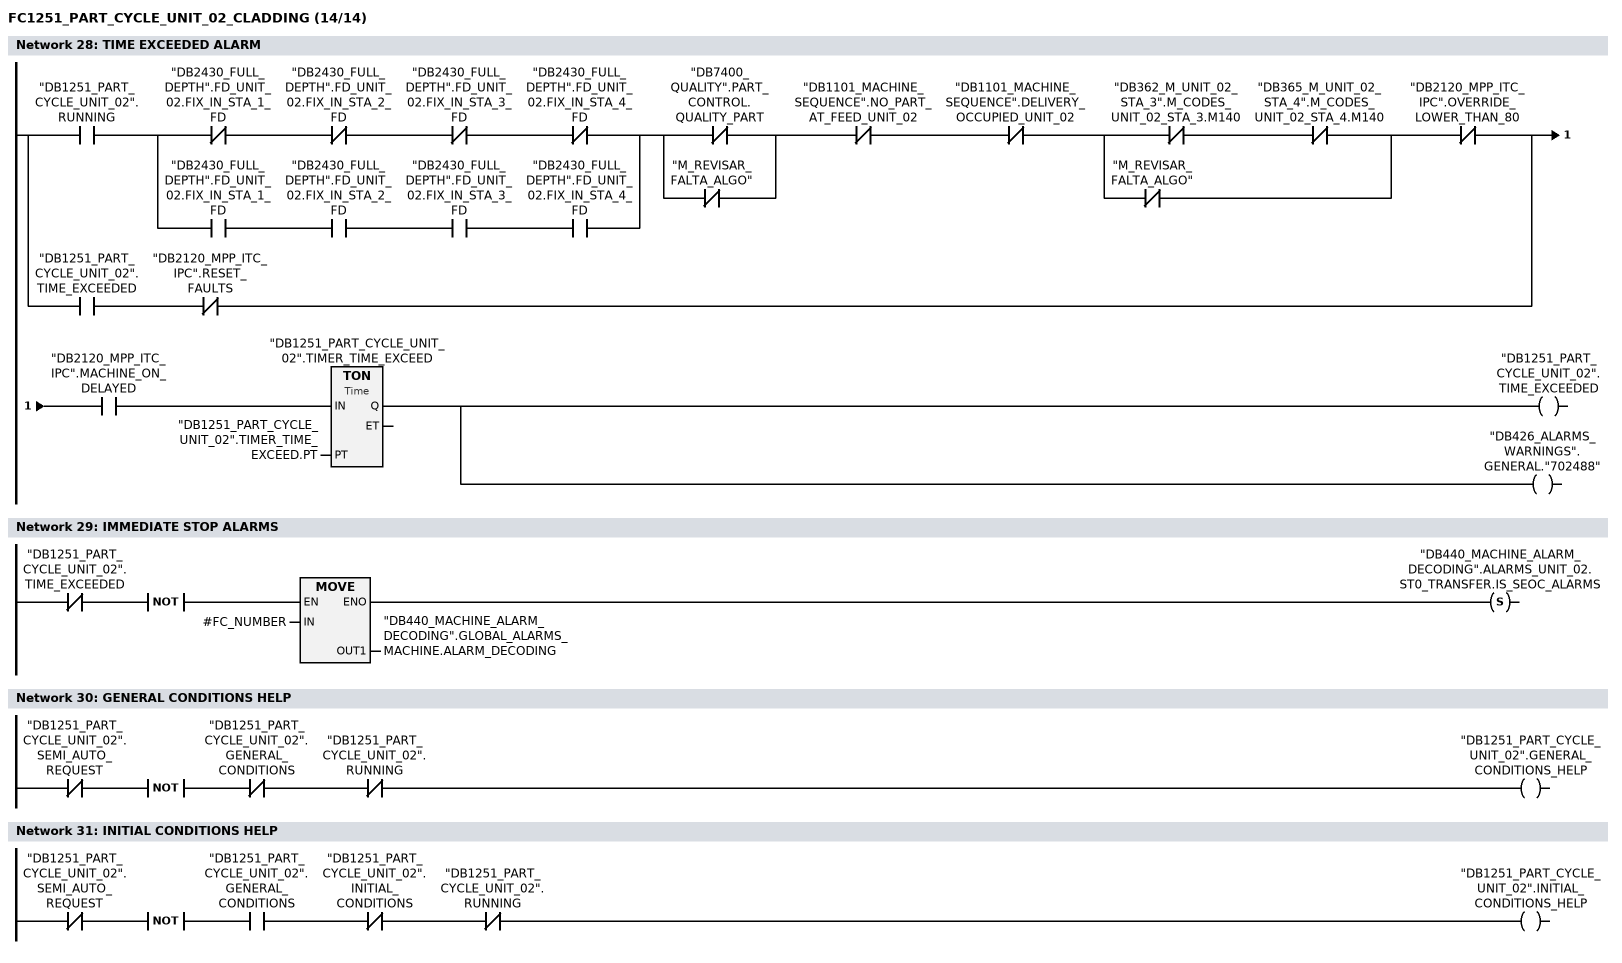
   RUNG wire#powerrail
      Contact( "DB1251_PART_CYCLE_UNIT_02".RUNNING )
      wire#w1
      I_Contact( "DB2430_FULL_DEPTH".FD_UNIT_02.FIX_IN_STA_1_FD )
      I_Contact( "DB2430_FULL_DEPTH".FD_UNIT_02.FIX_IN_STA_2_FD )
      I_Contact( "DB2430_FULL_DEPTH".FD_UNIT_02.FIX_IN_STA_3_FD )
      I_Contact( "DB2430_FULL_DEPTH".FD_UNIT_02.FIX_IN_STA_4_FD )
      wire#w2
      I_Contact( "DB7400_QUALITY".PART_CONTROL.QUALITY_PART )
      wire#w3
      I_Contact( "DB1101_MACHINE_SEQUENCE".NO_PART_AT_FEED_UNIT_02 )
      I_Contact( "DB1101_MACHINE_SEQUENCE".DELIVERY_OCCUPIED_UNIT_02 )
      wire#w4
      I_Contact( "DB362_M_UNIT_02_STA_3".M_CODES_UNIT_02_STA_3.M140 )
      I_Contact( "DB365_M_UNIT_02_STA_4".M_CODES_UNIT_02_STA_4.M140 )
      wire#w5
      I_Contact( "DB2120_MPP_ITC_IPC".OVERRIDE_LOWER_THAN_80 )
      wire#w6
      Contact( "DB2120_MPP_ITC_IPC".MACHINE_ON_DELAYED )
      { S7_Templates := "time_type := Time" } "DB1251_PART_CYCLE_UNIT_02".TIMER_TIME_EXCEED.TON(pt := "DB1251_PART_CYCLE_UNIT_02".TIMER_TIME_EXCEED.PT, et =>)
      wire#w7
      Coil( "DB1251_PART_CYCLE_UNIT_02".TIME_EXCEEDED )
   END_RUNG
   RUNG wire#w1
      Contact( "DB2430_FULL_DEPTH".FD_UNIT_02.FIX_IN_STA_1_FD )
      Contact( "DB2430_FULL_DEPTH".FD_UNIT_02.FIX_IN_STA_2_FD )
      Contact( "DB2430_FULL_DEPTH".FD_UNIT_02.FIX_IN_STA_3_FD )
      Contact( "DB2430_FULL_DEPTH".FD_UNIT_02.FIX_IN_STA_4_FD )
   END_RUNG wire#w2
   RUNG wire#w2
      I_Contact( "M_REVISAR_FALTA_ALGO" )
   END_RUNG wire#w3
   RUNG wire#w4
      I_Contact( "M_REVISAR_FALTA_ALGO" )
   END_RUNG wire#w5
   RUNG wire#powerrail
      Contact( "DB1251_PART_CYCLE_UNIT_02".TIME_EXCEEDED )
      I_Contact( "DB2120_MPP_ITC_IPC".RESET_FAULTS )
   END_RUNG wire#w6
   RUNG wire#w7
      Coil( "DB426_ALARMS_WARNINGS".GENERAL."702488" )
   END_RUNG
   // the same network as SCL:
   "DB1251_PART_CYCLE_UNIT_02".TIMER_TIME_EXCEED.TON(IN := (("DB1251_PART_CYCLE_UNIT_02".RUNNING AND ((NOT "DB2430_FULL_DEPTH".FD_UNIT_02.FIX_IN_STA_1_FD AND NOT "DB2430_FULL_DEPTH".FD_UNIT_02.FIX_IN_STA_2_FD AND NOT "DB2430_FULL_DEPTH".FD_UNIT_02.FIX_IN_STA_3_FD AND NOT "DB2430_FULL_DEPTH".FD_UNIT_02.FIX_IN_STA_4_FD) OR ("DB2430_FULL_DEPTH".FD_UNIT_02.FIX_IN_STA_1_FD AND "DB2430_FULL_DEPTH".FD_UNIT_02.FIX_IN_STA_2_FD AND "DB2430_FULL_DEPTH".FD_UNIT_02.FIX_IN_STA_3_FD AND "DB2430_FULL_DEPTH".FD_UNIT_02.FIX_IN_STA_4_FD)) AND (NOT "DB7400_QUALITY".PART_CONTROL.QUALITY_PART OR NOT "M_REVISAR_FALTA_ALGO") AND NOT "DB1101_MACHINE_SEQUENCE".NO_PART_AT_FEED_UNIT_02 AND NOT "DB1101_MACHINE_SEQUENCE".DELIVERY_OCCUPIED_UNIT_02 AND ((NOT "DB362_M_UNIT_02_STA_3".M_CODES_UNIT_02_STA_3.M140 AND NOT "DB365_M_UNIT_02_STA_4".M_CODES_UNIT_02_STA_4.M140) OR NOT "M_REVISAR_FALTA_ALGO") AND NOT "DB2120_MPP_ITC_IPC".OVERRIDE_LOWER_THAN_80) OR ("DB1251_PART_CYCLE_UNIT_02".TIME_EXCEEDED AND NOT "DB2120_MPP_ITC_IPC".RESET_FAULTS)) AND "DB2120_MPP_ITC_IPC".MACHINE_ON_DELAYED,
                           PT := "DB1251_PART_CYCLE_UNIT_02".TIMER_TIME_EXCEED.PT);
   "DB1251_PART_CYCLE_UNIT_02".TIME_EXCEEDED := "DB1251_PART_CYCLE_UNIT_02".TIMER_TIME_EXCEED.Q;
   "DB426_ALARMS_WARNINGS".GENERAL."702488" := "DB1251_PART_CYCLE_UNIT_02".TIMER_TIME_EXCEED.Q;
END_REGION

REGION Network 29: IMMEDIATE STOP ALARMS
   RUNG wire#powerrail
      I_Contact( "DB1251_PART_CYCLE_UNIT_02".TIME_EXCEEDED )
      Not()
      { S7_GenerateENO := "TRUE" } Move(in := #FC_NUMBER, out1 => "DB440_MACHINE_ALARM_DECODING".GLOBAL_ALARMS_MACHINE.ALARM_DECODING)
      S_Coil( "DB440_MACHINE_ALARM_DECODING".ALARMS_UNIT_02.ST0_TRANSFER.IS_SEOC_ALARMS )
   END_RUNG
   // the same network as SCL:
   // ENO of a box is taken as its EN; it also drops when the box reports an error
   IF NOT (NOT "DB1251_PART_CYCLE_UNIT_02".TIME_EXCEEDED) THEN
       "DB440_MACHINE_ALARM_DECODING".GLOBAL_ALARMS_MACHINE.ALARM_DECODING := #FC_NUMBER;
       "DB440_MACHINE_ALARM_DECODING".ALARMS_UNIT_02.ST0_TRANSFER.IS_SEOC_ALARMS := TRUE;
   END_IF;
END_REGION

REGION Network 30: GENERAL CONDITIONS HELP
   RUNG wire#powerrail
      I_Contact( "DB1251_PART_CYCLE_UNIT_02".SEMI_AUTO_REQUEST )
      Not()
      I_Contact( "DB1251_PART_CYCLE_UNIT_02".GENERAL_CONDITIONS )
      I_Contact( "DB1251_PART_CYCLE_UNIT_02".RUNNING )
      Coil( "DB1251_PART_CYCLE_UNIT_02".GENERAL_CONDITIONS_HELP )
   END_RUNG
   // the same network as SCL:
   "DB1251_PART_CYCLE_UNIT_02".GENERAL_CONDITIONS_HELP := NOT (NOT "DB1251_PART_CYCLE_UNIT_02".SEMI_AUTO_REQUEST) AND NOT "DB1251_PART_CYCLE_UNIT_02".GENERAL_CONDITIONS AND NOT "DB1251_PART_CYCLE_UNIT_02".RUNNING;
END_REGION

REGION Network 31: INITIAL CONDITIONS HELP
   RUNG wire#powerrail
      I_Contact( "DB1251_PART_CYCLE_UNIT_02".SEMI_AUTO_REQUEST )
      Not()
      Contact( "DB1251_PART_CYCLE_UNIT_02".GENERAL_CONDITIONS )
      I_Contact( "DB1251_PART_CYCLE_UNIT_02".INITIAL_CONDITIONS )
      I_Contact( "DB1251_PART_CYCLE_UNIT_02".RUNNING )
      Coil( "DB1251_PART_CYCLE_UNIT_02".INITIAL_CONDITIONS_HELP )
   END_RUNG
   // the same network as SCL:
   "DB1251_PART_CYCLE_UNIT_02".INITIAL_CONDITIONS_HELP := NOT (NOT "DB1251_PART_CYCLE_UNIT_02".SEMI_AUTO_REQUEST) AND "DB1251_PART_CYCLE_UNIT_02".GENERAL_CONDITIONS AND NOT "DB1251_PART_CYCLE_UNIT_02".INITIAL_CONDITIONS AND NOT "DB1251_PART_CYCLE_UNIT_02".RUNNING;
END_REGION
END_FUNCTION
